(* CODESYS project OC_Profinet.library
   DefaultNamespace: OC_Profinet
   DocFormat: reStructuredText
   Description: Open Commissioning Library for Profinet devices
   Author: SpiraTec AG
   Title: OC_Profinet
   Version: 0.0.1
   Company: Open Commissioning
   Placeholder: OC_Profinet

Project tree, tasks and I/O mapping:
  libraries: OC_Core, * (Open Commissioning); Tc2_Math, * (Beckhoff Automation GmbH); Tc2_Standard, * (Beckhoff Automation GmbH); Tc2_System, * (Beckhoff Automation GmbH); Tc2_Utilities, * (Beckhoff Automation GmbH); Tc3_Module, * (Beckhoff Automation GmbH); TcUnit, * (www.tcunit.org)
  Common/
    ProfidriveBaseState/
    ProfidriveParamInterpreter/
      data type E_ProfidriveParamFormat
      function block FB_ProfidriveParamInterpreter [ST]: FormatSize, FormatType, MakeResponse, Reset
      data type ST_ProfidriveParam
      data type ST_ProfidriveParamSet
  Devices/
    Communication/
      RcvDp/
        function block FB_RcvDp [ST]: AssignProcessData, ControlLogic, InitRun, ReadBus, SimLogic, WriteBus
        data type ST_RcvDpConfig
        data type ST_RcvDpCtrl
        data type ST_RcvDpDevData
        data type ST_RcvDpHstData
        data type ST_RcvDpStatus
      SendDp/
        function block FB_SendDp [ST]: AssignProcessData, ControlLogic, InitRun, PlcAddress, ReadBus, SimLogic, WriteBus
        data type ST_SendDpConfig
        data type ST_SendDpCtrl
        data type ST_SendDpDevData
        data type ST_SendDpHstData
        data type ST_SendDpStatus
      function F_CalcCrc16 [ST]
    Drives/
      MoviCPosition/
        data type E_MoviCPositionOperationMode
        function block FB_MoviCPosition [ST]: AssignProcessData, ControlLogic, GetControlData, InitRun, Operation, Safety, SetStatusData
        data type ST_MoviCPosition_Config
        data type ST_MoviCPosition_Control
        data type ST_MoviCPosition_Status
      MoviCVelocity/
        function block FB_MoviCVelocity [ST]: AssignProcessData, ControlLogic, GetControlData, InitRun, Operation, Safety, SetStatusData
        data type ST_MoviCVelocity_Config
        data type ST_MoviCVelocity_Control
        data type ST_MoviCVelocity_Status
      MovisafeCSBx1a/
        function block FB_MovisafeCSBx1a [ST]: AssignProcessData, ControlLogic, GetControlData, InitRun, SetStatusData
        data type ST_MovisafeCSBx1a_Config
        data type ST_MovisafeCSBx1a_Control
        data type ST_MovisafeCSBx1a_Status
      MovisafeCSSx1a/
        function block FB_MovisafeCSSx1a [ST]: AssignProcessData, ControlLogic, GetControlData, InitRun, SetStatusData
        data type ST_MovisafeCSSx1a_Config
        data type ST_MovisafeCSSx1a_Control
        data type ST_MovisafeCSSx1a_Status
      ProfidriveGSM/
        data type E_ProfidriveGSM_State
        function block FB_ProfidriveGSM [ST]: eState, nControl, nStatus, S0_Disabled, S1_SwitchingOnInhibited, S2_ReadyForSwitchingOn, S3_SwitchedOn, S4_Operation, S51_RampStop, S52_QuickStop
        data type ST_ProfiidriveGSM_STW1
        data type ST_ProfiidriveGSM_ZSW1
      ProfidriveTelegram1/
        function block FB_ProfidriveTelegram1 [ST]: AssignProcessData, ControlLogic, GetControlData, InitRun, Operation, SetStatusData
        data type ST_ProfidriveTelegram1_Config
        data type ST_ProfidriveTelegram1_Control
        data type ST_ProfidriveTelegram1_Status
  Tests/
    Drives/
      function block FB_ProfidriveGSM_Test [ST]: TestState_S0, TestState_S1, TestState_S2, TestState_S3, TestState_S4, TestState_S51, TestState_S52, TestTransitions_S0, TestTransitions_S1, TestTransitions_S2, TestTransitions_S3, TestTransitions_S4, TestTransitions_S51, TestTransitions_S52
      function block FB_ProfidriveTelegram1_Test [ST]: Test_ProcessDataControl, Test_ProcessDataStatus
    program PRG_TEST [ST]
*)

// Common/ProfidriveParamInterpreter/E_ProfidriveParamFormat
{attribute 'qualified_only'}
{attribute 'strict'}
{attribute 'conditionalshow'}
TYPE E_ProfidriveParamFormat :
(
	UNKNOWN := 0,
	INT8	:= 2,
	INT16	:= 3,
	INT32	:= 4,
	UINT8	:= 5,
	UINT16	:= 6,
	UINT32	:= 7,
	FLOAT	:= 8,
	ZERO	:= 64,
	BYTE_	:= 65,
	WORD_	:= 66,
	DWORD_	:= 67,
	ERROR	:= 68
) BYTE;
END_TYPE

// Common/ProfidriveParamInterpreter/ST_ProfidriveParam
{attribute 'conditionalshow'}
TYPE ST_ProfidriveParam :
STRUCT
	nAttribute	: BYTE;
	nNumber		: UINT;
	nSubIndex	: UINT;
	nElements	: BYTE;
	nFormat		: E_ProfidriveParamFormat;
	aValue		: ARRAY[0..234] OF BYTE;
END_STRUCT
END_TYPE

// Common/ProfidriveParamInterpreter/ST_ProfidriveParamSet
{attribute 'conditionalshow'}
TYPE ST_ProfidriveParamSet :
	ARRAY[0..22] OF ST_ProfidriveParam; 
END_TYPE

// Devices/Communication/RcvDp/ST_RcvDpConfig
TYPE ST_RcvDpConfig :
STRUCT
	nDpDpId			 			: UINT := 0;
	fTimeout		 			: REAL := 0.5;
	bAutoAckRei					: BOOL := TRUE;
END_STRUCT
END_TYPE

// Devices/Communication/RcvDp/ST_RcvDpCtrl
{attribute 'pack_mode' := '1'}
TYPE ST_RcvDpCtrl :
STRUCT
	nRcvBoolData			: WORD;
	nRcvInt00				: INT;
	nRcvInt01				: INT;
	nRcvData				: WORD;
	nRcvSequenceNumber		: WORD;
	nRcvCrc					: WORD;
END_STRUCT
END_TYPE

// Devices/Communication/RcvDp/ST_RcvDpDevData
TYPE ST_RcvDpDevData :
STRUCT
	bAckRei		: BOOL;
	bSub00		: BOOL;
	bSub01		: BOOL;
	bSub02		: BOOL;
	bSub03		: BOOL;
	bSub04		: BOOL;
	bSub05		: BOOL;
	bSub06		: BOOL;
	bSub07		: BOOL;
	bSub08		: BOOL;
	bSub09		: BOOL;
	bSub10		: BOOL;
	bSub11		: BOOL;
	bSub12		: BOOL;
	bSub13		: BOOL;
	bSub14		: BOOL;
	bSub15		: BOOL;
	nSub00		: INT;
	nSub01		: INT;
END_STRUCT
END_TYPE

// Devices/Communication/RcvDp/ST_RcvDpHstData
TYPE ST_RcvDpHstData :
STRUCT
	bError		: BOOL;
	bSubsOn		: BOOL;
	bRcv00		: BOOL;
	bRcv01		: BOOL;
	bRcv02		: BOOL;
	bRcv03		: BOOL;
	bRcv04		: BOOL;
	bRcv05		: BOOL;
	bRcv06		: BOOL;
	bRcv07		: BOOL;
	bRcv08		: BOOL;
	bRcv09		: BOOL;
	bRcv10		: BOOL;
	bRcv11		: BOOL;
	bRcv12		: BOOL;
	bRcv13		: BOOL;
	bRcv14		: BOOL;
	bRcv15		: BOOL;
	nRcv00		: INT;
	nRcv01		: INT;
END_STRUCT
END_TYPE

// Devices/Communication/RcvDp/ST_RcvDpStatus
{attribute 'pack_mode' := '1'}
TYPE ST_RcvDpStatus :
STRUCT
	nSendData				: WORD;
	nSendSequenceNumber		: WORD;	
	nSendCrc				: WORD;
END_STRUCT
END_TYPE

// Devices/Communication/SendDp/ST_SendDpConfig
TYPE ST_SendDpConfig :
STRUCT
	nDpDpId			 			: UINT := 0;
	fTimeout		 			: REAL := 0.5;
END_STRUCT
END_TYPE

// Devices/Communication/SendDp/ST_SendDpCtrl
TYPE ST_SendDpCtrl :
STRUCT
	nRcvData				: WORD;
	nRcvSequenceNumber		: WORD;	
	nRcvCrc					: WORD;
END_STRUCT
END_TYPE

// Devices/Communication/SendDp/ST_SendDpDevData
TYPE ST_SendDpDevData :
STRUCT
	bSend00		: BOOL;
	bSend01		: BOOL;
	bSend02		: BOOL;
	bSend03		: BOOL;
	bSend04		: BOOL;
	bSend05		: BOOL;
	bSend06		: BOOL;
	bSend07		: BOOL;
	bSend08		: BOOL;
	bSend09		: BOOL;
	bSend10		: BOOL;
	bSend11		: BOOL;
	bSend12		: BOOL;
	bSend13		: BOOL;
	bSend14		: BOOL;
	bSend15		: BOOL;
	nSend00		: INT;
	nSend01		: INT;
END_STRUCT
END_TYPE

// Devices/Communication/SendDp/ST_SendDpHstData
TYPE ST_SendDpHstData :
STRUCT
	bError		: BOOL;
	bSubsOn		: BOOL;
END_STRUCT
END_TYPE

// Devices/Communication/SendDp/ST_SendDpStatus
TYPE ST_SendDpStatus :
STRUCT
	nSendBoolData			: WORD;
	nSendInt00				: INT;
	nSendInt01				: INT;
	nSendData				: WORD;
	nSendSequenceNumber		: WORD;
	nSendCrc				: WORD;
END_STRUCT
END_TYPE

// Devices/Drives/MoviCPosition/E_MoviCPositionOperationMode
{attribute 'qualified_only'}
TYPE E_MoviCPositionOperationMode :
(
	Jog					:= 100, //Position controlled jogging
	JogNoEnc			:= 101, //Speed controlled jogging
	SpeedControl		:= 200, //Speed control
	ReferenceParam		:= 300, //Reference travel, offset via parameter
	ReferenceBus		:= 301, //Reference travel, offset via fieldbus
	PositionAbs			:= 400, //Absolute position control
	PositionRel			:= 401, //Relative position control
	PositionModPos		:= 402, //Modulo position control, positive
	PositionModNeg		:= 403, //Modulo position control, negative
	PositionModShort	:= 404, //Modulo position control, shortest distance
	EnergyOptimized		:= 1200, //Energieoptimiertes Positionieren
	MechanicsOptimized	:= 1210	 //Mechanikoptimiertes Positionieren
)INT;
END_TYPE

// Devices/Drives/MoviCPosition/ST_MoviCPosition_Config
TYPE ST_MoviCPosition_Config :
STRUCT
	pMovisafeCSSx1a			: POINTER TO FB_MovisafeCSSx1a; //[optional] Pointer to a MovisafeCSSx1a instance
	nSoftwareLimitMin		: DINT := -2147483648;	//Position limit minimum in LU
	nSoftwareLimitMax		: DINT := 2147483647;	//Position limit maximum in LU
	nReferencePos			: DINT := 0;			//Reference position in LU when using mode 300
	fDecCoastStop			: REAL := 1000.0;		//Deceleration for coast/brake stop in LU/s^2
	fDecEstop				: REAL := 100.0;		//Deceleration for emergency stop in LU/s^2
	fDecelerationLimit		: REAL := 100.0;		//Decceleration limit (bus stop) in LU/s^2
	fRatioVelocity			: REAL := 1.0;			//Ratio for setpoint velocity
	fRatioAccDec			: REAL := 1.0;			//Ratio for setpoint acceleration/deceleration
	fRatioPosition			: REAL := 1.0;			//Ratio for position output
	nJerk					: INT  := 0;			//Jerk from 0 to 100%
	fPositionOffset			: REAL := 0;
	fInitPosition			: REAL := 0;
	fResolution				: REAL := 0.1;
	bSwapProcessData		: BOOL; //SWAP Process Data from/to FIELDBUS
END_STRUCT
END_TYPE

// Devices/Drives/MoviCPosition/ST_MoviCPosition_Control
{attribute 'pack_mode' := '1'}
TYPE ST_MoviCPosition_Control :
STRUCT
    b0_EnableEStop 					: BIT;	//0  1 = enable, 0 = emergency stop
    b1_EnableBusStop 				: BIT;	//1  1 = enable, 0 = stop at application limits
    b2_Reserved2 					: BIT;	//2
    b3_ReleaseBrake 				: BIT;	//3  only needed if function is activated
    b4_JoggingCW 					: BIT;	//4  jog positive
    b5_JoggingCCW 					: BIT;	//5  jog negative
    b6_AcceptRelativePosition 		: BIT;	//6  apply relative target pos only in relative pos mode
    b7_StartStop 					: BIT;	//7  1 = start movement in all modes except jog, 0 = deceleration to speed 0
    b8_ErrorReset 					: BIT;	//8  reset fault messages
    b9_Reserved9 					: BIT;	//9
    b10_ActivateDriveTrain2 		: BIT;	//10  0 = drive train 1 selected, 1 = drive train 2 selected
    b11_Reserved11 					: BIT;	//11
    b12_DisableSoftwareLimits 		: BIT;	//12  0 = software limit activated, 1 = software limit deactivated
    b13_ActivateInhibit 			: BIT;	//13  1 = output stage inhibit activated -> motor coasts to halt or brake is applied, 0 = output stage can be enabled
    b14_ActivateStandByMode 		: BIT;	//14  1 = activated, can only be activated when output stage is inhibited (bActivateInhibit = 1)
    b15_MovikitHeartbeat 			: BIT;	//15  Heartbeat trigger
	nSetpointSpeed					: INT;	//16..31 
	nSetpointAcceleration			: INT;	//32..47
	nSetpointDeceleration			: INT;	//48..63
	nDigitalOutputs					: WORD;	//64..79
	nTargetApplicationMode			: E_MoviCPositionOperationMode; //80..95
	nTargetPosition					: DINT;	//96..127
END_STRUCT
END_TYPE

// Devices/Drives/MoviCPosition/ST_MoviCPosition_Status
{attribute 'pack_mode' := '1'}
TYPE ST_MoviCPosition_Status :
STRUCT
	b0_InverterReady					: BIT;	//0  1 = Ready
	b1_STOInactive						: BIT;	//1  1 = STO inactive
	b2_PowerStageOn						: BIT;	//2  1 = Output stage enable
	b3_BrakeReleased					: BIT;	//3  1 = Brake released
	b4_MotorTurning						: BIT;	//4  1 = Motor running
	b5_DriveReferenced					: BIT;	//5  1 = Active drive referenced
	b6_SetpointsActive					: BIT;	//6  1 = New relative position applied
	b7_TargetpositionReached			: BIT;	//7  1 = In position
	b8_ErrorActive						: BIT;	//8  1 = Fault
	b9_WarningActive					: BIT;	//9  1 = Warning
	b10_DriveTrain2Active				: BIT;	//10  1 = Drive train 2 active
	b11_SpeedSetpointReached			: BIT;	//11  1 = "Setpoint/actual speed comparison active" signal
	b12_SoftwareLimitsDisabled			: BIT;	//12  1 = Software limit switches inactive
	b13_OutputStageInhibit 				: BIT;	//13  1 = Output stage inhibit 
	b14_StandByModeActive				: BIT;	//14  1 = Standby mode active
	b15_MovikitHeartbeat				: BIT;	//15  Heartbeat trigger mirror
	nActualSpeed						: INT;	//16..31
	nActualStatus						: WORD;	//32..47
	nActualTorque						: INT;	//48..63
	nDigitalInputs						: WORD;	//64..79
	nActualApplicationMode				: E_MoviCPositionOperationMode; //80..95
	nActualPosition						: DINT;	//96..127 
END_STRUCT
END_TYPE

// Devices/Drives/MoviCVelocity/ST_MoviCVelocity_Config
TYPE ST_MoviCVelocity_Config :
STRUCT
	pMovisafeCSSx1a			: POINTER TO FB_MovisafeCSSx1a; //[optional] Pointer to a MovisafeCSSx1a instance
	nSoftwareLimitMin		: DINT := -2147483648;	//Position limit minimum in LU
	nSoftwareLimitMax		: DINT := 2147483647;	//Position limit maximum in LU
	nReferencePos			: DINT := 0;			//Reference position in LU when using mode 300
	fDecCoastStop			: REAL := 1000.0;		//Deceleration for coast/brake stop in LU/s^2
	fDecEstop				: REAL := 100.0;		//Deceleration for emergency stop in LU/s^2
	fDecelerationLimit		: REAL := 100.0;		//Decceleration limit (bus stop) in LU/s^2
	fRatioVelocity			: REAL := 1.0;			//Ratio for setpoint velocity
	fRatioAccDec			: REAL := 1.0;			//Ratio for setpoint acceleration/deceleration
	fRatioPosition			: REAL := 1.0;			//Ratio for position output
	nJerk					: INT  := 0;			//Jerk from 0 to 100%
	fPositionOffset			: REAL := 0;
	fInitPosition			: REAL := 0;
	fResolution				: REAL := 0.1;
	bSwapProcessData		: BOOL; //SWAP Process Data from/to FIELDBUS
	bOutputVelocity			: BOOL := TRUE;		//TRUE: TargetValue = Velocity, FALSE: TargetValue = Position
END_STRUCT
END_TYPE

// Devices/Drives/MoviCVelocity/ST_MoviCVelocity_Control
TYPE ST_MoviCVelocity_Control :
STRUCT
    b0_EnableEStop 					: BIT;	//0  1 = enable, 0 = emergency stop
    b1_EnableBusStop 				: BIT;	//1  1 = enable, 0 = stop at application limits
    b2_Reserved2 					: BIT;	//2
    b3_ReleaseBrake 				: BIT;	//3  only needed if function is activated
    b4_JoggingCW 					: BIT;	//4  jog positive
    b5_JoggingCCW 					: BIT;	//5  jog negative
    b6_AcceptRelativePosition 		: BIT;	//6  apply relative target pos only in relative pos mode
    b7_StartStop 					: BIT;	//7  1 = start movement in all modes except jog, 0 = deceleration to speed 0
    b8_ErrorReset 					: BIT;	//8  reset fault messages
    b9_Reserved9 					: BIT;	//9
    b10_ActivateDriveTrain2 		: BIT;	//10  0 = drive train 1 selected, 1 = drive train 2 selected
    b11_Reserved11 					: BIT;	//11
    b12_DisableSoftwareLimits 		: BIT;	//12  0 = software limit activated, 1 = software limit deactivated
    b13_ActivateInhibit 			: BIT;	//13  1 = output stage inhibit activated -> motor coasts to halt or brake is applied, 0 = output stage can be enabled
    b14_ActivateStandByMode 		: BIT;	//14  1 = activated, can only be activated when output stage is inhibited (bActivateInhibit = 1)
    b15_MovikitHeartbeat 			: BIT;	//15  Heartbeat trigger
	nSetpointSpeed					: INT;	//16..31 
	nSetpointAcceleration			: INT;	//32..47
	nSetpointDeceleration			: INT;	//48..63
	nDigitalOutputs					: WORD;	//64..79	
END_STRUCT
END_TYPE

// Devices/Drives/MoviCVelocity/ST_MoviCVelocity_Status
{attribute 'pack_mode' := '1'}
TYPE ST_MoviCVelocity_Status :
STRUCT
	b0_InverterReady					: BIT;	//0  1 = Ready
	b1_STOInactive						: BIT;	//1  1 = STO inactive
	b2_PowerStageOn						: BIT;	//2  1 = Output stage enable
	b3_BrakeReleased					: BIT;	//3  1 = Brake released
	b4_MotorTurning						: BIT;	//4  1 = Motor running
	b5_DriveReferenced					: BIT;	//5  1 = Active drive referenced
	b6_SetpointsActive					: BIT;	//6  1 = New relative position applied
	b7_TargetpositionReached			: BIT;	//7  1 = In position
	b8_ErrorActive						: BIT;	//8  1 = Fault
	b9_WarningActive					: BIT;	//9  1 = Warning
	b10_DriveTrain2Active				: BIT;	//10  1 = Drive train 2 active
	b11_SpeedSetpointReached			: BIT;	//11  1 = "Setpoint/actual speed comparison active" signal
	b12_SoftwareLimitsDisabled			: BIT;	//12  1 = Software limit switches inactive
	b13_OutputStageInhibit 				: BIT;	//13  1 = Output stage inhibit 
	b14_StandByModeActive				: BIT;	//14  1 = Standby mode active
	b15_MovikitHeartbeat				: BIT;	//15  Heartbeat trigger mirror
	nActualSpeed						: INT;	//16..31
	nActualStatus						: WORD;	//32..47
	nActualTorque						: INT;	//48..63
	nDigitalInputs						: WORD;	//64..79	
END_STRUCT
END_TYPE

// Devices/Drives/MovisafeCSBx1a/ST_MovisafeCSBx1a_Config
TYPE ST_MovisafeCSBx1a_Config :
STRUCT	
	bSwapProcessData		: BOOL; //SWAP Process Data from/to FIELDBUS
END_STRUCT
END_TYPE

// Devices/Drives/MovisafeCSBx1a/ST_MovisafeCSBx1a_Control
{attribute 'pack_mode' := '1'}
TYPE ST_MovisafeCSBx1a_Control :
STRUCT
	b0_STO1				: BIT; //Sicher abgeschaltetes Drehmoment
	b1_Reserve			: BIT; //Reserve
	b2_Reserve			: BIT; //Reserve
	b3_Reserve			: BIT; //Reserve
	b4_Reserve			: BIT; //Reserve
	b5_Reserve			: BIT; //Reserve
	bQUIT_F_DI			: BIT; //Quittierung der verriegelten Digitaleingänge
	bQUIT_ERROR			: BIT; //Quittierung der Fehler Sicherheitskarte
	b8_Reserve			: BIT; //Reserve
	b9_Reserve			: BIT; //Reserve
	b10_Reserve			: BIT; //Reserve
	b11_Reserve			: BIT; //Reserve
	b12_Reserve			: BIT; //Reserve
	b13_Reserve			: BIT; //Reserve
	b14_Reserve			: BIT; //Reserve
	b15_Reserve			: BIT; //Reserve
	b16_Reserve			: BIT; //Reserve
	b17_Reserve			: BIT; //Reserve
	b18_SSx1			: BIT; //Antriebssicherheitsfunktion SSx1 deaktivieren
	b19_SSx2			: BIT; //Antriebssicherheitsfunktion SSx2 deaktivieren
	b20_Reserve			: BIT; //Reserve
	b21_Reserve			: BIT; //Reserve
	b22_Reserve			: BIT; //Reserve
	b23_Reserve			: BIT; //Reserve
END_STRUCT
END_TYPE

// Devices/Drives/MovisafeCSBx1a/ST_MovisafeCSBx1a_Status
{attribute 'pack_mode' := '1'}
TYPE ST_MovisafeCSBx1a_Status :
STRUCT
	b0_STO_ACTIVE		: BIT; //Sicher abgeschaltetes Drehmoment
	b1_Reserve			: BIT; //Reserve
	b2_Reserve			: BIT; //Reserve
	b3_INPUT_DATA_VALID	: BIT; //Alle Prozesswerte der F-DI enthalten aktuelle Werte
	b4_Reserve			: BIT; //Reserve
	b5_Reserve			: BIT; //Reserve
	b6_WARNING			: BIT; //Warnung in der Safety-option
	b7_ERROR_STATE		: BIT; //Fehler in der Safety-option
	b8_F_DI0			: BIT; //Zustand digitaler Eingang 1
	b9_F_DI1			: BIT; //Zustand digitaler Eingang 2
	b10_F_DI2			: BIT; //Zustand digitaler Eingang 3
	b11_F_DI3			: BIT; //Zustand digitaler Eingang 4
	b12_Reserve			: BIT; //Reserve
	b13_Reserve			: BIT; //Reserve
	b14_Reserve			: BIT; //Reserve
	b15_Reserve			: BIT; //Reserve
	b16_Reserve			: BIT; //Reserve
	b17_Reserve			: BIT; //Reserve
	b18_SSx1			: BIT; //SSx1  ist aktiviert
	b19_SSx2			: BIT; //SSx2 ist aktiviert
	b20_Reserve			: BIT; //Reserve
	b21_Reserve			: BIT; //Reserve
	b22_Reserve			: BIT; //Reserve
	b23_Reserve			: BIT; //Reserve
	b24_Reserve			: BIT; //Reserve
	b25_Reserve			: BIT; //Reserve
	b26_Reserve			: BIT; //Reserve
	b27_Reserve			: BIT; //Reserve
	b28_Reserve			: BIT; //Reserve
	b29_Reserve			: BIT; //Reserve
	b30_Reserve			: BIT; //Reserve
	b31_Reserve			: BIT; //Reserve
END_STRUCT
END_TYPE

// Devices/Drives/MovisafeCSSx1a/ST_MovisafeCSSx1a_Config
TYPE ST_MovisafeCSSx1a_Config :
STRUCT	
	bSwapProcessData		: BOOL; //SWAP Process Data from/to FIELDBUS
END_STRUCT
END_TYPE

// Devices/Drives/MovisafeCSSx1a/ST_MovisafeCSSx1a_Control
{attribute 'pack_mode' := '1'}
TYPE ST_MovisafeCSSx1a_Control :
STRUCT
	bSTO				: BIT; //0.0  Sicher abgeschaltetes Drehmoment
	bSLI				: BIT; //0.1  Freigabe SLI (Sicher begrenztes Schrittmaß)
	bSBT				: BIT; //0.2  Freigabe SBT (Sicherer Bremsentest)
	bRES_3				: BIT; //0.3  Reserve
	bMUTING_ENC_ERR		: BIT; //0.4  Muting Geber anwählen
	bTEST_MODE_ACTIVE	: BIT; //0.5  Test Modus der Antriebssicherheitsfunktion anwählen
	bQUIT_F_DI			: BIT; //0.6  Quittierung der verriegelten Digitaleingänge
	bQUIT_ERROR			: BIT; //0.7  Quittierung der Fehler Sicherheitskarte
	bF_DO_0				: BIT; //1.0  F-DO 00 Digitaler Ausgang 0
	bF_DO_1				: BIT; //1.1  F-DO 01 Digitaler Ausgang 1
	bRES_12				: BIT; //1.2  Reserve
	bRES_13				: BIT; //1.3  Reserve
	bRES_14				: BIT; //1.4  Reserve
	bRES_15				: BIT; //1.5  Reserve
	bRES_16				: BIT; //1.6  Reserve
	bRES_17				: BIT; //1.7  Reserve
	bSOS_1				: BIT; //2.0  SOS1 deaktivieren (Sicherer Betriebshalt)
	bRES_21				: BIT; //2.1  Reserve
	bSSx1				: BIT; //2.2  Antriebssicherheitsfunktion SSx1 deaktivieren
	bSSx2				: BIT; //2.3  Antriebssicherheitsfunktion SSx2 deaktivieren
	bSDI_1				: BIT; //2.4  SDI 1 deaktivieren (Sichere Bewegungsrichtung)
	bSDI_2				: BIT; //2.5  SDI 2 deaktivieren (Sichere Bewegungsrichtung)
	bSLI_1				: BIT; //2.6  SLI 1 deaktivieren (Sicher begrenztes Schrittmaß)
	bSLI_2				: BIT; //2.7  SLI 2 deaktivieren (Sicher begrenztes Schrittmaß)
	bSLS_1				: BIT; //3.0  SLS 1 deaktivieren (Sicher begrenzte Geschwindigkeit)
	bSLS_2				: BIT; //3.1  SLS 2 deaktivieren (Sicher begrenzte Geschwindigkeit)
	bSLS_3				: BIT; //3.2  SLS 3 deaktivieren (Sicher begrenzte Geschwindigkeit)
	bSLS_4				: BIT; //3.3  SLS 4 deaktivieren (Sicher begrenzte Geschwindigkeit)
	bSSR_1				: BIT; //3.4  SSR 1 deaktivieren (Sicherer Geschwindigkeitsbereich)
	bSSR_2				: BIT; //3.5  SSR 2 deaktivieren (Sicherer Geschwindigkeitsbereich)
	bRES_36				: BIT; //3.6  Reserve
	bRES_37				: BIT; //3.7  Reserve
	bSLA_1				: BIT; //4.0  SLA 1 deaktivieren (Sicher begrenzte Beschleunigung)
	bSLA_2				: BIT; //4.1  SLA 2 deaktivieren (Sicher begrenzte Beschleunigung)
	bRES_42				: BIT; //4.2  Reserve
	bRES_43				: BIT; //4.3  Reserve
	bRES_44				: BIT; //4.4  Reserve
	bRES_45				: BIT; //4.5  Reserve
	bRES_46				: BIT; //4.6  Reserve
	bRES_47				: BIT; //4.7  Reserve
END_STRUCT
END_TYPE

// Devices/Drives/MovisafeCSSx1a/ST_MovisafeCSSx1a_Status
{attribute 'pack_mode' := '1'}
TYPE ST_MovisafeCSSx1a_Status :
STRUCT
	bSTO_ACTIVE			: BIT; //0.0  Sicher abgeschaltetes Drehmoment
	bASF_DIAG			: BIT; //0.1  Mindestens eine Antriebssicherheitsfunktion hat eine Grenze überschritten
	bSBT_ACTIVE			: BIT; //0.2  Bremsentest ist aktiv
	bINPUT_DATA_VALID	: BIT; //0.3  Alle Prozesswerte der F-DI enthalten aktuelle Werte
	bMUTING_ENC_ERR		: BIT; //0.4  Geber Muting Funktion ist aktive
	bTEST_MODE_ACTIVE	: BIT; //0.5  Test Modus der Antriebssicherheitsfunktion ist aktive
	bWARNING			: BIT; //0.6  Warnung in der Safety-option
	bERROR_STATE		: BIT; //0.7  Fehler in der Safety-option
	bF_DI0				: BIT; //1.0  Zustand digitaler Eingang 1
	bF_DI1				: BIT; //1.1  Zustand digitaler Eingang 2
	bF_DI2				: BIT; //1.2  Zustand digitaler Eingang 3
	bF_DI3				: BIT; //1.3  Zustand digitaler Eingang 4
	bRES_14				: BIT; //1.4  Reserve
	bRES_15				: BIT; //1.5  Reserve
	bRES_16				: BIT; //1.6  Reserve
	bRES_17				: BIT; //1.7  Reserve
	bSOS_1				: BIT; //2.0  SOS1 ist aktiviert (Sicherer Betriebshalt)
	bRES_21				: BIT; //2.1  Reserve
	bSSx1				: BIT; //2.2  SSx1  ist aktiviert
	bSSx2				: BIT; //2.3  SSx2 ist aktiviert
	bSDI_1				: BIT; //2.4  SDI 1  ist aktiviert (Sichere Bewegungsrichtung)
	bSDI_2				: BIT; //2.5  SDI 2  ist aktiviert (Sichere Bewegungsrichtung)
	bSLI_1				: BIT; //2.6  SLI 1  ist aktiviert (Sicher begrenztes Schrittmaß)
	bSLI_2				: BIT; //2.7  SLI 2  ist aktiviert (Sicher begrenztes Schrittmaß)
	bSLS_1				: BIT; //3.0  SLS 1  ist aktiviert (Sicher begrenzte Geschwindigkeit)
	bSLS_2				: BIT; //3.1  SLS 2  ist aktiviert (Sicher begrenzte Geschwindigkeit)
	bSLS_3				: BIT; //3.2  SLS 3  ist aktiviert (Sicher begrenzte Geschwindigkeit)
	bSLS_4				: BIT; //3.3  SLS 4  ist aktiviert (Sicher begrenzte Geschwindigkeit)
	bSSR_1				: BIT; //3.4  SSR 1  ist aktiviert (Sicherer Geschwindigkeitsbereich)
	bSSR_2				: BIT; //3.5  SSR 2  ist aktiviert (Sicherer Geschwindigkeitsbereich)
	bRES_36				: BIT; //3.6  Reserve
	bRES_37				: BIT; //3.7  Reserve
	bSLA_1				: BIT; //4.0  SLA 1  ist aktiviert (Sicher begrenzte Beschleunigung)
	bSLA_2				: BIT; //4.1  SLA 2  ist aktiviert (Sicher begrenzte Beschleunigung)
	bSSM_1				: BIT; //4.2  SSM 1  ist aktiviert (Sichere Geschwindigkeitsüberwachung)
	bSSM_2				: BIT; //4.3  SSM 2  ist aktiviert (Sichere Geschwindigkeitsüberwachung)
	bSSM_3				: BIT; //4.4  SSM 3  ist aktiviert (Sichere Geschwindigkeitsüberwachung)
	bSSM_4				: BIT; //4.5  SSM 4  ist aktiviert (Sichere Geschwindigkeitsüberwachung)
	bRES_46				: BIT; //4.6  Reserve
	bRES_47				: BIT; //4.7  Reserve
	bRES_50				: BIT; //5.0  Reserve
	bRES_51				: BIT; //5.1  Reserve
	bRES_52				: BIT; //5.2  Reserve
	bRES_53				: BIT; //5.3  Reserve
	bRES_54				: BIT; //5.4  Reserve
	bRES_55				: BIT; //5.5  Reserve
	bRES_56				: BIT; //5.6  Reserve
	bRES_57				: BIT; //5.7  Reserve
END_STRUCT
END_TYPE

// Devices/Drives/ProfidriveGSM/E_ProfidriveGSM_State
{attribute 'qualified_only'}
{attribute 'strict'}
{attribute 'conditionalshow'}
TYPE E_ProfidriveGSM_State :
(
	S0_Disabled := 0,
	S1_SwitchingOnInhibited := 1,
	S2_ReadyForSwitchingOn := 2,
	S3_SwitchedOn := 3,
	S4_Operation := 4,
	S51_RampStop := 51,
	S52_QuickStop := 52
);
END_TYPE

// Devices/Drives/ProfidriveGSM/ST_ProfiidriveGSM_STW1
{attribute 'pack_mode' := '1'}
TYPE ST_ProfiidriveGSM_STW1 :
STRUCT
	b0_On 							: BIT; 	//ON/OFF (OFF1)
	b1_CoastStop					: BIT; 	//The axis will not coast stop if this bit is set (OFF2)
	b2_QuickStop					: BIT; 	//The axis will not execute quick stop if this bit is set. Quick stop executes a controlled stop on the axis. (OFF3)
	b3_EnableOperation				: BIT; 	//The axis will enable and execute command if all preconditions are set. If a Wake and Shake procedure has to be executed as part of enabling, the transition to state "S4: Operation Enabled" is delayed until the procedure is finished.
	b4_Reserve						: BIT;	//Reserve
	b5_Reserve						: BIT;	//Reserve
	b6_Reserve						: BIT;	//Reserve
	b7_FaultAcknowledge				: BIT;	//Set this bit to reset faults on the drive.
	b8_Reserve						: BIT;	//Reserve
	b9_Reserve						: BIT;	//Reserve	
	b10_ControlPlc					: BIT;	//When not set, no command is accepted from the PLC.	
	b11_Reserved					: BIT;	//Reserve
	b12_Reserved					: BIT;	//Reserve
	b13_Reserved					: BIT;	//Reserve
	b14_Reserved					: BIT;	//Reserve
	b15_Reserved					: BIT;	//Reserve
END_STRUCT
END_TYPE

// Devices/Drives/ProfidriveGSM/ST_ProfiidriveGSM_ZSW1
{attribute 'pack_mode' := '1'}
TYPE ST_ProfiidriveGSM_ZSW1 :
STRUCT
	b0_ReadyToSwitchOn 				: BIT; 	//Ready to switch on
	b1_ReadyForOperation			: BIT; 	//Ready for operation
	b2_OperationEnabled				: BIT; 	//Operation enabled
	b3_FaultPresent					: BIT; 	//A fault is present on the axis
	b4_CoastStop 					: BIT;	//No coast stop is executed (No OFF2 is active)
	b5_QuickStop					: BIT;	//No quick stop is executed (No OFF3 is active)
	b6_SwitchingOnInhibited			: BIT;	//Switch-on inhibit Switching on again is only possible through OFF1 and subsequent ON.
	b7_WarningPresent				: BIT;	//Warning present. The drive is operating. No acknowledgment required
	b8_Reserve						: BIT;	//Reserve
	b9_ControlRequested				: BIT;	//Control requested by the master
	b10_Reserved					: BIT;	//Reserve
	b11_Reserved					: BIT;	//Reserve
	b12_Reserved					: BIT;	//Reserve
	b13_Reserved					: BIT;	//Reserve
	b14_Reserved					: BIT;	//Reserve
	b15_Reserved					: BIT;	//Reserve
END_STRUCT
END_TYPE

// Devices/Drives/ProfidriveTelegram1/ST_ProfidriveTelegram1_Config
TYPE ST_ProfidriveTelegram1_Config :
STRUCT
	fRampDownTimeCoastStop 		: REAL := 1.0;		//Coast stop deceleration time in s
	bControlRequested			: BOOL := TRUE;
	bOutputVelocity				: BOOL := TRUE;		//TRUE: TargetValue = Velocity, FALSE: TargetValue = Position
	fP1058						: REAL := 150.0;	//JOG 1 velocity in rotation/s
	fP1059						: REAL := -150.0;	//JOG 1 velocity in rotation/s
	fP1120						: REAL := 2.0;		//Default acceleration time in s
	fP1121						: REAL := 2.0;		//Default deceleration time in s
	fP1135						: REAL := 1.0;		//Ramp down time quick stop in s
	fP2000						: REAL := 3000;		//Velocity in rotation/s when targeting 16#4000
	nR0035						: REAL := 60.0; 	//Temperature in degree celcius	
	bSwapProcessData			: BOOL; //SWAP Process Data from/to FIELDBUS
END_STRUCT
END_TYPE

// Devices/Drives/ProfidriveTelegram1/ST_ProfidriveTelegram1_Control
TYPE ST_ProfidriveTelegram1_Control :
STRUCT
	b0_OFF1								: BOOL;	//STW1_0	0 = OFF1 (braking with ramp-function generator, then pulse suppression & ready for switching on) | 0 → 1 = ON (pulses can be enabled)
	b1_OFF2								: BOOL;	//STW1_1	0 = OFF2 (immediate pulse suppression and switching on inhibited) | 1 = No OFF2 (enable is possible)
	b2_OFF3								: BOOL;	//STW1_2	0 = OFF3 (braking with the OFF3 ramp p1135, then pulse suppression and switching on inhibited) | 1 = No OFF3 (enable possible) 
	b3_EnableOperation					: BOOL;	//STW1_3	0 = Inhibit operation (suppress pulses) | 1 = Enable operation (pulses can be enabled) 
	b4_OperatingCondition				: BOOL;	//STW1_4	0 = Inhibit ramp-function generator (set the ramp-function generator output to zero) | 1 = Operating condition (the ramp-function generator can be enabled)
	b5_ContinueRampFunctionGenerator	: BOOL;	//STW1_5	0 = Freeze ramp-function generator (freeze the ramp-function generator output) | 1 = Continue ramp-function generator 
	b6_EnableSetpoint  					: BOOL;	//STW1_6	0 = Inhibit setpoint (set the ramp-function generator input to zero) | 1 = Enable setpoint 
	b7_AcknowledgeFaults				: BOOL;	//STW1_7	0 → 1: = Acknowledge faults	                            
	b8_Jog1								: BOOL;	//STW1_8	1 = Jog 1 signal source
	b9_Jog2								: BOOL;	//STW1_9	1 = Jog 2 signal source
	b10_ControlByPLC					: BOOL;	//STW1_10	1 = Control by PLC
	b11_SetpointInversion				: BOOL;	//STW1_11	1 = Setpoint inversion
	b12_Reserved						: BOOL;	//STW1_12	Reserved
	b13_PotentiometerSetpointRaise		: BOOL;	//STW1_13	1 = Motorized potentiometer setpoint raise
	b14_PotentiometerSetpointLower		: BOOL;	//STW1_14	1 = Motorized potentiometer setpoint lower
	b15_Reserved						: BOOL;	//STW1_15	Reserved	
	nNSoll 								: INT;
END_STRUCT
END_TYPE

// Devices/Drives/ProfidriveTelegram1/ST_ProfidriveTelegram1_Status
TYPE ST_ProfidriveTelegram1_Status :
STRUCT
	b0_ReadyForSwitchingOn				: BOOL; // ZSW1_0	1 = Ready for switching on
	b1_ReadyForOperation				: BOOL; // ZSW1_1	1 = Ready for operation
	b2_OperationEnabled					: BOOL; // ZSW1_2	1 = Operation enabled
	b3_FaultPresent						: BOOL; // ZSW1_3	1 = Fault present
	b4_NoCoastDownActive				: BOOL; // ZSW1_4	1 = No coast down active (OFF2 inactive)
	b5_NoQuickStopActive				: BOOL; // ZSW1_5	1 = No quick stop active (OFF3 inactive)
	b6_SwitchingOnInhibited				: BOOL; // ZSW1_6	1 = Switching on inhibited active
	b7_AlarmPresent						: BOOL; // ZSW1_7	1 = Alarm present                        	
	b8_DeviationWithinTolerance			: BOOL; // ZSW1_8	1 = Speed setpoint - actual value deviation within tolerance t_off
	b9_ControlRequested					: BOOL; // ZSW1_9	1 = Control requested        
	b10_RpmCompValueReachedOrExceeded	: BOOL; // ZSW1_10	1 = f or n comparison value reached/exceeded  
	b11_TorqueOrPowerLimitNotReached	: BOOL; // ZSW1_11	1 = I, M, or P limit not reached     
	b12_OpenHoldingBrake 				: BOOL; // ZSW1_12	1 = Open the holding brake      
	b13_NoOvertempAlarm					: BOOL; // ZSW1_13	1 = No motor overtemperature alarm      
	b14_MotorRotatesForwards			: BOOL; // ZSW1_14	1 = Motor rotates forwards (n_act >= 0) | 0 = Motor rotates backwards (n_act < 0)   
	b15_NoAlarmNoOvertempPowerUnit		: BOOL; // ZSW1_15	1 = No alarm, thermal overload, power unit  
	nNIst								: INT;
END_STRUCT
END_TYPE

// Common/ProfidriveParamInterpreter/FB_ProfidriveParamInterpreter
FUNCTION_BLOCK INTERNAL FB_ProfidriveParamInterpreter
VAR_INPUT
	(* Pointer to raw user data *)
	pRawData		: POINTER TO BYTE;
	(* Pointer to array of parameters *)
	pParamSet		: POINTER TO ST_ProfidriveParamSet;
END_VAR
VAR_OUTPUT
	(* Reference number for response *)
	nReference		: BYTE;
	(* 1 = read, 2 = write *)
	nCommand		: BYTE;
	(* Addressed axis number *)
	nAxis			: BYTE;
	(* Number of parameters to read/write *)
	nParameters		: BYTE;
END_VAR
VAR
	nOffsReq		: BYTE;
	nOffsValue		: BYTE;
	nFormatSize		: BYTE;
	nValues			: BYTE;
	i, j, k			: UINT;
END_VAR

(* Copy header (first 4 bytes) *)
	nReference := pRawData[0];
	nCommand := pRawData[1];
	nAxis := pRawData[2];
	nParameters := pRawData[3];

(* Set request offset behind header *)
	nOffsReq := 4;

(* Set value offset behind last request *)
	nOffsValue := 4 + nParameters * 6;

(* Reset all parameters *)
	memset(pParamSet, 0, SIZEOF(ST_PROFIdriveParamSet));

(* Check parameter number *)	
	IF nParameters = 0 THEN
		RETURN;
	END_IF

(* Loop through number of parameter requests *)
	FOR i := 0 TO nParameters - 1 BY 1 DO
		
		(* Get parameter request information (6 bytes)... *)
		pParamSet^[i].nAttribute := pRawData[nOffsReq];
		pParamSet^[i].nElements := pRawData[nOffsReq + 1];
		pParamSet^[i].nNumber := pRawData[nOffsReq + 2] * 16#100 + pRawData[nOffsReq + 3];
		pParamSet^[i].nSubIndex := pRawData[nOffsReq + 4] * 16#100 + pRawData[nOffsReq + 5];
		
		(* ... and set offset to next request *)
		nOffsReq := nOffsReq + 6;
				
		(* Write command -> get values *)
		IF nCommand = 2 THEN		
			(* Get format *)
			nFormatSize := FormatSize(pRawData[nOffsValue]);
			pParamSet^[i].nFormat := FormatType(pRawData[nOffsValue]);
			nOffsValue := nOffsValue + 1;
			
			(* Get number of values *)
			nValues := pRawData[nOffsValue];
			nOffsValue := nOffsValue + 1;
			
			(* Loop through number of values *)
			FOR j := 0 TO nValues - 1 BY 1 DO
				
				(* Set value offset behind current values *)
				nOffsValue := nOffsValue + nFormatSize;
				
				(* Loop through format size and get values in reverse order *)
				FOR k := 0 TO nFormatSize - 1 BY 1 DO
					pParamSet^[i].aValue[j + k] := pRawData[nOffsValue - k - 1];
				END_FOR
			END_FOR
			
			(* Check if odd and set to even number *)
			IF nOffsValue.0 THEN
				nOffsValue := nOffsValue + 1;
			END_IF
		END_IF
	END_FOR

METHOD INTERNAL FormatSize : BYTE
VAR_INPUT
	nFormat	: BYTE;
END_VAR
CASE nFormat OF
	 16#02 : FormatSize := 2;
	 16#03 : FormatSize := 2;
	 16#04 : FormatSize := 4;
	 16#05 : FormatSize := 2;
	 16#06 : FormatSize := 2;
	 16#07 : FormatSize := 4;
	 16#08 : FormatSize := 4;
	 16#40 : FormatSize := 0;
	 16#41 : FormatSize := 2;
	 16#42 : FormatSize := 2;
	 16#43 : FormatSize := 4;
	 16#44 : FormatSize := 0;
ELSE
	FormatSize := 0;
END_CASE
END_METHOD

METHOD INTERNAL FormatType : E_ProfidriveParamFormat
VAR_INPUT
	nFormat	: BYTE;
END_VAR
CASE nFormat OF
	 16#02 : FormatType := E_ProfidriveParamFormat.INT8;
	 16#03 : FormatType := E_ProfidriveParamFormat.INT16;
	 16#04 : FormatType := E_ProfidriveParamFormat.INT32;
	 16#05 : FormatType := E_ProfidriveParamFormat.UINT8;
	 16#06 : FormatType := E_ProfidriveParamFormat.UINT16;
	 16#07 : FormatType := E_ProfidriveParamFormat.UINT32;
	 16#08 : FormatType := E_ProfidriveParamFormat.FLOAT;
	 16#40 : FormatType := E_ProfidriveParamFormat.ZERO;
	 16#41 : FormatType := E_ProfidriveParamFormat.BYTE_;
	 16#42 : FormatType := E_ProfidriveParamFormat.WORD_;
	 16#43 : FormatType := E_ProfidriveParamFormat.DWORD_;
	 16#44 : FormatType := E_ProfidriveParamFormat.ERROR;
ELSE
	FormatType := E_PROFIdriveParamFormat.UNKNOWN;
END_CASE
END_METHOD

METHOD INTERNAL MakeResponse : BOOL
VAR_INPUT
	(* Pointer to acyclic user data *)
	pResData		: POINTER TO BYTE;
END_VAR
VAR
	nOffset			: BYTE;
	nFormatSize		: BYTE;
	i, j, k			: UINT;
END_VAR
(* Copy header (first 4 bytes) *)
	pResData[0] := nReference;
	pResData[1] := nCommand;
	pResData[2] := nAxis;
	pResData[3] := nParameters;

(* Set offset behind header *)
	nOffset := 4;
	
(* Check parameter number *)	
	IF nParameters = 0 THEN
		RETURN;
	END_IF

(* Loop through number of parameter requests *)
	FOR i := 0 TO nParameters - 1 BY 1 DO
		
		(* Set format *)
		pResData[nOffset] := pParamSet^[i].nFormat;
		nFormatSize := FormatSize(pParamSet^[i].nFormat);
		nOffset := nOffset + 1;
		
		(* Set number of values *)
		pResData[nOffset] := pParamSet^[i].nElements;
		nOffset := nOffset + 1;
		
		(* Loop through number of elements *)
		FOR j := 0 TO pParamSet^[i].nElements - 1 BY 1 DO
			
			(* Set value offset behind current values *)
			nOffset := nOffset + nFormatSize;
			
			(* Loop through format size and get values in reverse order *)
			
			IF nFormatSize > 0 THEN
				FOR k := 0 TO nFormatSize - 1 BY 1 DO
					pResData[nOffset - k - 1] := pParamSet^[i].aValue[j + k] ;
				END_FOR
			END_IF
			
		END_FOR
		
		(* Check if odd and set to even number *)
		IF nOffset.0 THEN
			nOffset := nOffset + 1;
		END_IF	
	END_FOR

(* Return true when finished *)
	MakeResponse := TRUE;
END_METHOD

METHOD INTERNAL Reset : BOOL
nReference := 0;
nCommand := 0;
nAxis := 0;
nParameters := 0;
memset(pParamSet, 0, SIZEOF(ST_ProfidriveParamSet));
END_METHOD

END_FUNCTION_BLOCK

// Devices/Communication/RcvDp/FB_RcvDp
{attribute 'reflection'} 
FUNCTION_BLOCK FB_RcvDp EXTENDS FB_Base
VAR_INPUT
	stDevData			: ST_RcvDpDevData;
	stConfig 			: ST_RcvDpConfig;
END_VAR

VAR_OUTPUT
	stHstData			: ST_RcvDpHstData;
END_VAR

VAR
    {attribute 'instance-path'} 
    {attribute 'noinit'} 
    sPath 				: STRING; 
	pControlData		: POINTER TO BYTE;
	pStatusData			: POINTER TO BYTE;
	stCtrl				: ST_RcvDpCtrl; 
	stStatus			: ST_RcvDpStatus; 
	nLastSequenceNumber	: WORD;
	nCalculatedCrc		: WORD;	
	TonTimeout			: TON;	
END_VAR

VAR CONSTANT
	nPolynom			: WORD := 16#4EAB;
END_VAR

SUPER^();
InitRun();	
ReadBus();
ControlLogic();
WriteBus();

(*Assign Process Data Objects to device*)
METHOD PUBLIC AssignProcessData : BOOL
VAR_INPUT
	aControlData 		: ANY; //Addr. Process Output 12 bytes
	aStatusData 		: ANY; //Addr. Process Input 6 bytes
END_VAR
THIS^.pControlData := aControlData.pValue;
THIS^.pStatusData := aStatusData.pValue;
END_METHOD

METHOD INTERNAL ControlLogic
VAR_INPUT
END_VAR
(* Simplified communication when using PLCSIM Adv. *)
	IF OC_Core.GVL_Core.fbSystem.eControllerType = E_ControllerType.PlcSimAdvanced THEN
		SimLogic();
		RETURN;
	END_IF

(* Calculate received crc *)
	nCalculatedCrc := F_CalcCrc16(ADR(stCtrl), 8, stConfig.nDpDpId, nPolynom);

(* Restart timer, if sequence number has changed *)
	IF stCtrl.nRcvSequenceNumber <> nLastSequenceNumber AND NOT stHstData.bError THEN
		nLastSequenceNumber := stCtrl.nRcvSequenceNumber;
		stHstData.bSubsOn	:= FALSE;
		TonTimeout.IN		:= FALSE;
	ELSE
		TonTimeout.IN		:= TRUE;
	END_IF

(* Reintegration *)
	IF (stConfig.bAutoAckRei AND stHstData.bError) OR stDevData.bAckRei THEN
		stHstData.bError 	:= FALSE;
		TonTimeout.IN		:= FALSE;
	END_IF

(* Check if timer has expired *)
	TonTimeout();
	
	IF TonTimeout.Q	THEN
		stHstData.bError	:= TRUE;
		stHstData.bSubsOn	:= TRUE;
	END_IF

(* compare received crc value with calculated crc *)
	IF stCtrl.nRcvCrc = nCalculatedCrc AND NOT stHstData.bError THEN
		stHstData.bSubsOn	:= FALSE;
	ELSE
		stHstData.bError	:= TRUE;
		stHstData.bSubsOn	:= TRUE;
	END_IF

(* Get substitude or safety values *)
	IF stHstData.bSubsOn THEN
		stHstData.bRcv00	:= stDevData.bSub00;
		stHstData.bRcv01	:= stDevData.bSub01;
		stHstData.bRcv02	:= stDevData.bSub02;
		stHstData.bRcv03	:= stDevData.bSub03;
		stHstData.bRcv04	:= stDevData.bSub04;
		stHstData.bRcv05	:= stDevData.bSub05;
		stHstData.bRcv06	:= stDevData.bSub06;
		stHstData.bRcv07	:= stDevData.bSub07;
		stHstData.bRcv08	:= stDevData.bSub08;
		stHstData.bRcv09	:= stDevData.bSub09;
		stHstData.bRcv10	:= stDevData.bSub10;
		stHstData.bRcv11	:= stDevData.bSub11;
		stHstData.bRcv12	:= stDevData.bSub12;
		stHstData.bRcv13	:= stDevData.bSub13;
		stHstData.bRcv14	:= stDevData.bSub14;
		stHstData.bRcv15	:= stDevData.bSub15;
		stHstData.nRcv00	:= stDevData.nSub00;
		stHstData.nRcv01	:= stDevData.nSub01;
	ELSE
		stHstData.bRcv00	:= stCtrl.nRcvBoolData.0;
		stHstData.bRcv01	:= stCtrl.nRcvBoolData.1;
		stHstData.bRcv02	:= stCtrl.nRcvBoolData.2;
		stHstData.bRcv03	:= stCtrl.nRcvBoolData.3;
		stHstData.bRcv04	:= stCtrl.nRcvBoolData.4;
		stHstData.bRcv05	:= stCtrl.nRcvBoolData.5;
		stHstData.bRcv06	:= stCtrl.nRcvBoolData.6;
		stHstData.bRcv07	:= stCtrl.nRcvBoolData.7;
		stHstData.bRcv08	:= stCtrl.nRcvBoolData.8;  
		stHstData.bRcv09	:= stCtrl.nRcvBoolData.9;  
		stHstData.bRcv10	:= stCtrl.nRcvBoolData.10;  
		stHstData.bRcv11	:= stCtrl.nRcvBoolData.11;  
		stHstData.bRcv12	:= stCtrl.nRcvBoolData.12; 
		stHstData.bRcv13	:= stCtrl.nRcvBoolData.13; 
		stHstData.bRcv14	:= stCtrl.nRcvBoolData.14; 
		stHstData.bRcv15	:= stCtrl.nRcvBoolData.15;	
		stHstData.nRcv00	:= stCtrl.nRcvInt00;
		stHstData.nRcv01	:= stCtrl.nRcvInt01;
	END_IF

(* Send data *)
	stStatus.nSendData				:= BOOL_TO_WORD(stHstData.bSubsOn);
	stStatus.nSendSequenceNumber	:= stCtrl.nRcvSequenceNumber;
	stStatus.nSendCrc 				:= F_CalcCrc16(ADR(stStatus.nSendData), 2, stConfig.nDpDpId, nPolynom);
END_METHOD

METHOD INTERNAL InitRun : BOOL
VAR_INST
	bInitRun : BOOL := TRUE;
END_VAR
IF NOT bInitRun THEN RETURN; END_IF
bInitRun := FALSE;

IF pControlData = 0 OR pStatusData = 0 THEN
	ADSLOGSTR(ADSLOG_MSGTYPE_WARN, CONCAT(sPath, ': %s'), 'Plc address not set.');
END_IF

TonTimeout.PT := REAL_TO_TIME(stConfig.fTimeout);
END_METHOD

METHOD INTERNAL ReadBus
VAR_INPUT
END_VAR
IF pControlData = 0 THEN
	RETURN;
END_IF

stCtrl.nRcvBoolData 		:= pControlData[0] + pControlData[1] * 16#100;
stCtrl.nRcvInt00 			:= UINT_TO_INT(pControlData[2] * 16#100 + pControlData[3]);
stCtrl.nRcvInt01 			:= UINT_TO_INT(pControlData[4] * 16#100 + pControlData[5]);
stCtrl.nRcvData 			:= pControlData[6] + pControlData[7] * 16#100;
stCtrl.nRcvSequenceNumber 	:= pControlData[8] * 16#100 + pControlData[9];
stCtrl.nRcvCrc 				:= pControlData[10] * 16#100 + pControlData[11];
END_METHOD

METHOD INTERNAL SimLogic
VAR_INPUT
END_VAR
(* No error or substitude values in sim mode *)
	stHstData.bError 	:= FALSE;
	stHstData.bSubsOn	:= FALSE;

(* Get safety values *)
	stHstData.bRcv00	:= stCtrl.nRcvBoolData.0;
	stHstData.bRcv01	:= stCtrl.nRcvBoolData.1;
	stHstData.bRcv02	:= stCtrl.nRcvBoolData.2;
	stHstData.bRcv03	:= stCtrl.nRcvBoolData.3;
	stHstData.bRcv04	:= stCtrl.nRcvBoolData.4;
	stHstData.bRcv05	:= stCtrl.nRcvBoolData.5;
	stHstData.bRcv06	:= stCtrl.nRcvBoolData.6;
	stHstData.bRcv07	:= stCtrl.nRcvBoolData.7;
	stHstData.bRcv08	:= stCtrl.nRcvBoolData.8;  
	stHstData.bRcv09	:= stCtrl.nRcvBoolData.9;  
	stHstData.bRcv10	:= stCtrl.nRcvBoolData.10;  
	stHstData.bRcv11	:= stCtrl.nRcvBoolData.11;  
	stHstData.bRcv12	:= stCtrl.nRcvBoolData.12; 
	stHstData.bRcv13	:= stCtrl.nRcvBoolData.13; 
	stHstData.bRcv14	:= stCtrl.nRcvBoolData.14; 
	stHstData.bRcv15	:= stCtrl.nRcvBoolData.15;	
	stHstData.nRcv00	:= stCtrl.nRcvInt00;
	stHstData.nRcv01	:= stCtrl.nRcvInt01;

(* Send data *)
	stStatus.nSendData				:= 16#80;
	stStatus.nSendSequenceNumber	:= stCtrl.nRcvSequenceNumber;
	stStatus.nSendCrc 				:= F_CalcCrc16(ADR(stStatus.nSendData), 2, stConfig.nDpDpId, nPolynom);
END_METHOD

METHOD INTERNAL WriteBus
VAR_INPUT
END_VAR
IF pStatusData = 0 THEN
	RETURN;
END_IF

memcpy(pStatusData, ADR(stStatus.nSendData), 2);
       
memcpy(pStatusData + 2, ADR(stStatus.nSendSequenceNumber) + 1, 1);
memcpy(pStatusData + 3, ADR(stStatus.nSendSequenceNumber), 1);
       
memcpy(pStatusData + 4, ADR(stStatus.nSendCrc) + 1, 1);
memcpy(pStatusData + 5, ADR(stStatus.nSendCrc), 1);
END_METHOD

END_FUNCTION_BLOCK

// Devices/Communication/F_CalcCrc16
FUNCTION F_CalcCrc16 : WORD
VAR_INPUT
	pData		: POINTER TO BYTE;
	nDataSize	: INT;
	nInitCRC	: WORD;
	nPolynom	: WORD;
END_VAR
VAR
	nCrc		: WORD;
	nDataX		: BYTE;
	nI			: INT;
	nJ			: INT;
END_VAR

nCrc := nInitCRC;

FOR nI := 0 TO nDataSize - 1 BY 1 DO
	nDataX	:= pData[nI];
	FOR nJ := 0 TO 7 BY 1 DO
		IF (SHR(nCrc,15) AND 1) <> (SHR(nDataX,7) AND 1) THEN
			nCrc := SHL(nCrc,1) XOR nPolynom;
		ELSE
			nCrc := SHL(nCrc,1);
		END_IF
		nDataX := SHL(nDataX,1);
	END_FOR	
END_FOR

F_CalcCrc16 := nCrc;

END_FUNCTION

// Devices/Communication/SendDp/FB_SendDp
{attribute 'reflection'} 
FUNCTION_BLOCK FB_SendDp EXTENDS FB_Base
VAR_INPUT
	stDevData			: ST_SendDpDevData;
	stConfig 			: ST_SendDpConfig;
END_VAR

VAR_OUTPUT
	stHstData			: ST_SendDpHstData;
END_VAR

VAR
    {attribute 'instance-path'} 
    {attribute 'noinit'} 
    sPath 				: STRING; 
	pControlData			: POINTER TO BYTE;
	pStatusData				: POINTER TO BYTE;
	stCtrl				: ST_SendDpCtrl; 
	stStatus			: ST_SendDpStatus; 
	nLastSequenceNumber	: WORD;
	nSendSequenceNumber	: WORD;
	nCalculatedCrc		: WORD;	
	TonTimeout			: TON;
END_VAR

VAR CONSTANT
	nPolynom			: WORD := 16#4EAB;
END_VAR

SUPER^();
InitRun();
ReadBus();
ControlLogic();
WriteBus();

(*Assign Process Data Objects to device*)
METHOD PUBLIC AssignProcessData : BOOL
VAR_INPUT
	aControlData 		: ANY; //Addr. Process Output 6 bytes
	aStatusData 		: ANY; //Addr. Process Input 12 bytes
END_VAR
THIS^.pControlData := aControlData.pValue;
THIS^.pStatusData := aStatusData.pValue;
END_METHOD

METHOD INTERNAL ControlLogic
(* Simplified communication when using PLCSIM Adv. *)
	IF OC_Core.GVL_Core.fbSystem.eControllerType = E_ControllerType.PlcSimAdvanced THEN
		SimLogic();
		RETURN;
	END_IF

(* Calculate received crc *)
	nCalculatedCrc := F_CalcCrc16(ADR(stCtrl), 2, stConfig.nDpDpId, nPolynom);

(* Restart timer, if sequence number has changed *)
	IF stCtrl.nRcvSequenceNumber <> nLastSequenceNumber THEN
		TonTimeout.IN		:= FALSE;
		nLastSequenceNumber := stCtrl.nRcvSequenceNumber;
		stHstData.bError	:= FALSE;
		stHstData.bSubsOn	:= FALSE;
	ELSE
		TonTimeout.IN		:= TRUE;
	END_IF

(* Check if timer has expired *)
	TonTimeout();
	
	IF TonTimeout.Q	THEN
		TonTimeout.IN		:= FALSE;
		nSendSequenceNumber := 0;
		stHstData.bError	:= TRUE;
		stHstData.bSubsOn	:= TRUE;
	END_IF

(* compare received crc value with calculated crc *)
	IF stCtrl.nRcvCrc = nCalculatedCrc THEN
		IF nSendSequenceNumber = stCtrl.nRcvSequenceNumber THEN
			IF nSendSequenceNumber = 0 THEN
				nSendSequenceNumber := 1;
			ELSE
				nSendSequenceNumber := nSendSequenceNumber + 1;
			END_IF
		END_IF
	END_IF

(* Limit sequence number to 32767 *)
	IF nSendSequenceNumber > 32767 THEN
		nSendSequenceNumber := 1;
	END_IF

(* Send data *)
	stStatus.nSendBoolData.0 		:= stDevData.bSend00;
	stStatus.nSendBoolData.1 		:= stDevData.bSend01;
	stStatus.nSendBoolData.2 		:= stDevData.bSend02;
	stStatus.nSendBoolData.3 		:= stDevData.bSend03;
	stStatus.nSendBoolData.4 		:= stDevData.bSend04;
	stStatus.nSendBoolData.5 		:= stDevData.bSend05;
	stStatus.nSendBoolData.6 		:= stDevData.bSend06;
	stStatus.nSendBoolData.7 		:= stDevData.bSend07;
	stStatus.nSendBoolData.8 		:= stDevData.bSend08;
	stStatus.nSendBoolData.9 		:= stDevData.bSend09;
	stStatus.nSendBoolData.10 		:= stDevData.bSend10;
	stStatus.nSendBoolData.11 		:= stDevData.bSend11;
	stStatus.nSendBoolData.12 		:= stDevData.bSend12;
	stStatus.nSendBoolData.13 		:= stDevData.bSend13;
	stStatus.nSendBoolData.14 		:= stDevData.bSend14;
	stStatus.nSendBoolData.15 		:= stDevData.bSend15;
	stStatus.nSendInt00				:= stDevData.nSend00;
	stStatus.nSendInt01				:= stDevData.nSend01;
	stStatus.nSendData				:= BOOL_TO_WORD(stHstData.bSubsOn);
	stStatus.nSendSequenceNumber 	:= nSendSequenceNumber;
	stStatus.nSendCrc 				:= F_CalcCrc16(ADR(stStatus), 8, stConfig.nDpDpId, nPolynom);
END_METHOD

METHOD INTERNAL InitRun : BOOL
VAR_INST
	bInitRun : BOOL := TRUE;
END_VAR
IF NOT bInitRun THEN RETURN; END_IF
bInitRun := FALSE;

IF pControlData = 0 OR pStatusData = 0 THEN
	ADSLOGSTR(ADSLOG_MSGTYPE_WARN, CONCAT(sPath, ': %s'), 'Plc address not set.');
END_IF

TonTimeout.PT := REAL_TO_TIME(stConfig.fTimeout);
END_METHOD

METHOD PUBLIC PlcAddress
VAR_INPUT
	I :	ANY; // Must be 6 bytes 
	Q :	ANY; // Must be 12 bytes
END_VAR
pControlData := Q.pValue;
pStatusData := I.pValue;
END_METHOD

METHOD INTERNAL ReadBus
VAR_INPUT
END_VAR
IF pControlData = 0 THEN
	RETURN;
END_IF

stCtrl.nRcvData 			:= pControlData[0] + pControlData[1] * 16#100;
stCtrl.nRcvSequenceNumber 	:= pControlData[2] * 16#100 + pControlData[3];
stCtrl.nRcvCrc 				:= pControlData[4] * 16#100 + pControlData[5];
END_METHOD

METHOD INTERNAL SimLogic
VAR_INPUT
END_VAR
(* No error or substitude values in sim mode *)
	stHstData.bError 	:= FALSE;
	stHstData.bSubsOn	:= FALSE;

(* Send data *)
	stStatus.nSendBoolData.0 		:= stDevData.bSend00;
	stStatus.nSendBoolData.1 		:= stDevData.bSend01;
	stStatus.nSendBoolData.2 		:= stDevData.bSend02;
	stStatus.nSendBoolData.3 		:= stDevData.bSend03;
	stStatus.nSendBoolData.4 		:= stDevData.bSend04;
	stStatus.nSendBoolData.5 		:= stDevData.bSend05;
	stStatus.nSendBoolData.6 		:= stDevData.bSend06;
	stStatus.nSendBoolData.7 		:= stDevData.bSend07;
	stStatus.nSendBoolData.8 		:= stDevData.bSend08;
	stStatus.nSendBoolData.9 		:= stDevData.bSend09;
	stStatus.nSendBoolData.10 		:= stDevData.bSend10;
	stStatus.nSendBoolData.11 		:= stDevData.bSend11;
	stStatus.nSendBoolData.12 		:= stDevData.bSend12;
	stStatus.nSendBoolData.13 		:= stDevData.bSend13;
	stStatus.nSendBoolData.14 		:= stDevData.bSend14;
	stStatus.nSendBoolData.15 		:= stDevData.bSend15;
	stStatus.nSendInt00				:= stDevData.nSend00;
	stStatus.nSendInt01				:= stDevData.nSend01;
	stStatus.nSendData				:= 16#80;
	stStatus.nSendSequenceNumber 	:= 16#FFFF;
	stStatus.nSendCrc 				:= F_CalcCrc16(ADR(stStatus), 8, stConfig.nDpDpId, nPolynom);
END_METHOD

METHOD INTERNAL WriteBus
VAR_INPUT
END_VAR
IF pStatusData = 0 THEN
	RETURN;
END_IF

memcpy(pStatusData, ADR(stStatus.nSendBoolData), 2);
       
memcpy(pStatusData + 2, ADR(stStatus.nSendInt00) + 1, 1);
memcpy(pStatusData + 3, ADR(stStatus.nSendInt00), 1);
       
memcpy(pStatusData + 4, ADR(stStatus.nSendInt01) + 1, 1);
memcpy(pStatusData + 5, ADR(stStatus.nSendInt01), 1);
              
memcpy(pStatusData + 6, ADR(stStatus.nSendData), 2);
              
memcpy(pStatusData + 8, ADR(stStatus.nSendSequenceNumber) + 1, 1);
memcpy(pStatusData + 9, ADR(stStatus.nSendSequenceNumber), 1);
               
memcpy(pStatusData + 10, ADR(stStatus.nSendCrc) + 1, 1);
memcpy(pStatusData + 11, ADR(stStatus.nSendCrc), 1);
END_METHOD

END_FUNCTION_BLOCK

// Devices/Drives/MoviCPosition/FB_MoviCPosition
{attribute 'reflection'}
FUNCTION_BLOCK FB_MoviCPosition EXTENDS FB_LinkDataReal
VAR_INPUT
	bSTO						: BOOL := TRUE;
	stControl 					: ST_MoviCPosition_Control;
	stConfig					: ST_MoviCPosition_Config;
	nDigitalInputs				: WORD;
END_VAR

VAR_OUTPUT
	stStatus					: ST_MoviCPosition_Status;
	fValue						: REAL;
END_VAR

VAR
    {attribute 'instance-path'} 
    {attribute 'noinit'} 
    sPath 						: STRING;	                			
	                			
	fbBaseState					: FB_ProfidriveGSM;
	fbBasicDrive				: FB_DriveControl;
	                				
	bOpModeValid				: BOOL;
	pMovisafe					: POINTER TO FB_MovisafeCSSx1a;	
	
	pControlData				: POINTER TO BYTE; //Addr. Process Output
	pStatusData					: POINTER TO BYTE; //Addr. Process Input
END_VAR

SUPER^();
InitRun();

GetControlData();
Safety();
ControlLogic();
SetStatusData();

(*Assign Process Data Objects to device*)
METHOD PUBLIC AssignProcessData : BOOL
VAR_INPUT
	aControlData 		: ANY; //Addr. Process Output
	aStatusData 		: ANY; //Addr. Process Input
END_VAR
THIS^.pControlData := aControlData.pValue;
THIS^.pStatusData := aStatusData.pValue;
END_METHOD

METHOD INTERNAL ControlLogic
//Unity Init - Load persistent data
IF SUPER^.Status.7 THEN
	IF stConfig.fRatioPosition <> 0 THEN	
		fbBasicDrive.fPosition := SUPER^.StatusData/stConfig.fRatioPosition - stConfig.fPositionOffset;
	ELSE
		fbBasicDrive.fPosition := SUPER^.StatusData - stConfig.fPositionOffset;
	END_IF
END_IF

(* Evaluate incoming operation mode *)
bOpModeValid := FALSE;

CASE stControl.nTargetApplicationMode OF
	E_MoviCPositionOperationMode.Jog:
		bOpModeValid := TRUE;
	E_MoviCPositionOperationMode.JogNoEnc:
		bOpModeValid := TRUE;
	E_MoviCPositionOperationMode.SpeedControl:
		bOpModeValid := TRUE;
	E_MoviCPositionOperationMode.ReferenceParam:
		bOpModeValid := TRUE;
	E_MoviCPositionOperationMode.ReferenceBus:
		bOpModeValid := TRUE;
	E_MoviCPositionOperationMode.PositionAbs, E_MoviCPositionOperationMode.EnergyOptimized, E_MoviCPositionOperationMode.MechanicsOptimized:
		bOpModeValid := TRUE;
	E_MoviCPositionOperationMode.PositionRel:
		bOpModeValid := TRUE;
	E_MoviCPositionOperationMode.PositionModPos:
		bOpModeValid := TRUE;
	E_MoviCPositionOperationMode.PositionModNeg:
		bOpModeValid := TRUE;
	E_MoviCPositionOperationMode.PositionModShort:
		bOpModeValid := TRUE;
END_CASE

(* Base state of the controller *)
fbBaseState.bStandstill := OC_Core.F_Compare(fbBasicDrive.fVelocity, 0, 1E-3);
fbBaseState.stSTW1.b0_On := stControl.b1_EnableBusStop AND fbBaseState.eState <> E_ProfidriveGSM_State.S1_SwitchingOnInhibited;
fbBaseState.stSTW1.b1_CoastStop := NOT stControl.b13_ActivateInhibit AND bSTO;
fbBaseState.stSTW1.b2_QuickStop := stControl.b0_EnableEStop;
fbBaseState.stSTW1.b3_EnableOperation := stControl.b7_StartStop AND bOpModeValid;

fbBaseState();
		
(* Set parameter of basic drive *)
IF stControl.b12_DisableSoftwareLimits THEN
	fbBasicDrive.fPositionLimitMin := -2147483648.0;
	fbBasicDrive.fPositionLimitMax := 2147483647.0;
	fbBasicDrive.fTolerance := 0.1;
ELSE
	fbBasicDrive.fPositionLimitMin := DINT_TO_REAL(stConfig.nSoftwareLimitMin);
	fbBasicDrive.fPositionLimitMax := DINT_TO_REAL(stConfig.nSoftwareLimitMax);
	fbBasicDrive.fTolerance := 0.1;
END_IF
					
(* Evaluate base state *)
CASE fbBaseState.eState OF
	
(* S1, S2 or S3 -> Drive coasts to a stop or brake is applied *)
	E_ProfidriveGSM_State.S1_SwitchingOnInhibited,
	E_ProfidriveGSM_State.S2_ReadyForSwitchingOn,
	E_ProfidriveGSM_State.S3_SwitchedOn:
		fbBasicDrive.Stop(stConfig.fDecCoastStop);

(* S4 -> Evaluate operation mode *)
	E_ProfidriveGSM_State.S4_Operation:
		Operation();

(* S5a -> Drive decelerates with application limit *)
	E_ProfidriveGSM_State.S51_RampStop:
		fbBasicDrive.Stop(stConfig.fDecelerationLimit);
		
(* S5b -> Drive decelerates with emergency stop ramp *)
	E_ProfidriveGSM_State.S52_QuickStop:
	    fbBasicDrive.Stop(stConfig.fDecEstop);
END_CASE
	
(* Status Word *)
stStatus.b0_InverterReady				:= TRUE;
stStatus.b1_STOInactive					:= bSTO;
stStatus.b2_PowerStageOn				:= stControl.b13_ActivateInhibit;
stStatus.b3_BrakeReleased				:= stControl.b1_EnableBusStop OR stControl.b3_ReleaseBrake;
stStatus.b4_MotorTurning				:= NOT fbBaseState.bStandstill;
stStatus.b5_DriveReferenced				:= TRUE;
stStatus.b6_SetpointsActive		 		:= FALSE;
stStatus.b7_TargetpositionReached		:= fbBasicDrive.bIsPositionReached;	
stStatus.b8_ErrorActive					:= FALSE;
stStatus.b9_WarningActive				:= FALSE;
stStatus.b10_DriveTrain2Active			:= stControl.b10_ActivateDriveTrain2;
stStatus.b11_SpeedSetpointReached		:= fbBasicDrive.bIsMoving;
stStatus.b12_SoftwareLimitsDisabled		:= stControl.b12_DisableSoftwareLimits;
stStatus.b13_OutputStageInhibit			:= fbBaseState.stZSW1.b6_SwitchingOnInhibited;
stStatus.b14_StandByModeActive			:= stControl.b14_ActivateStandByMode;
stStatus.b15_MovikitHeartbeat			:= stControl.b15_MovikitHeartbeat;

(* Status values *)
stStatus.nActualSpeed := REAL_TO_INT(fbBasicDrive.fVelocity / stConfig.fRatioVelocity);
stStatus.nActualStatus := 0;
stStatus.nActualTorque := 0;
stStatus.nDigitalInputs := nDigitalInputs;
IF bOpModeValid THEN
	stStatus.nActualApplicationMode := stControl.nTargetApplicationMode;
END_IF
stStatus.nActualPosition := REAL_TO_DINT(fbBasicDrive.fPosition);
	
(* Position output *)
THIS^.ControlData := fbBasicDrive.fPosition * stConfig.fRatioPosition + stConfig.fPositionOffset;
fValue := ControlData;
END_METHOD

METHOD INTERNAL GetControlData : BOOL
IF pControlData <= 0 THEN RETURN; END_IF

(* PO1 Control Word *)
F_Memcpy(ADR(stControl), pControlData, 2, stConfig.bSwapProcessData);
(* PO2 Setpoint Speed *)
F_Memcpy(ADR(stControl) + 2, pControlData + 2, 2, stConfig.bSwapProcessData);
(* PO3 Setpoint Acceleration *)
F_Memcpy(ADR(stControl) + 4, pControlData + 4, 2, stConfig.bSwapProcessData);
(* PO4 Setpoint Deceleration *)
F_Memcpy(ADR(stControl) + 6, pControlData + 6, 2, stConfig.bSwapProcessData);
(* PO5 Digital Outputs *)
F_Memcpy(ADR(stControl) + 8, pControlData + 8, 2, stConfig.bSwapProcessData);
(* PO6 Target Application Mode *)
F_Memcpy(ADR(stControl) + 10, pControlData + 10, 2, stConfig.bSwapProcessData);
(* PO7,PO8 Target Position *)
F_Memcpy(ADR(stControl) + 12, pControlData + 12, 4, stConfig.bSwapProcessData);
END_METHOD

METHOD INTERNAL InitRun
VAR_INST
	bInitRun : BOOL := TRUE;
END_VAR
IF NOT bInitRun THEN RETURN; END_IF
bInitRun := FALSE;

IF pControlData = 0 OR pStatusData = 0 THEN
	ADSLOGSTR(ADSLOG_MSGTYPE_WARN, CONCAT(sPath, ': %s'), 'Plc address not set.');
END_IF

pMovisafe := stConfig.pMovisafeCSSx1a;
fbBasicDrive.fPosition := stConfig.fInitPosition;
END_METHOD

METHOD INTERNAL Operation
VAR_INST
	fTargetPos			: REAL;
	fSetpointVel		: REAL;
	fSetpointAcc		: REAL;
	fSetpointDec		: REAL;
END_VAR
(* Copy setpoint values *)
fTargetPos 		:= DINT_TO_REAL(stControl.nTargetPosition);
fSetpointVel 	:= stControl.nSetpointSpeed * stConfig.fRatioVelocity; 
fSetpointAcc 	:= stControl.nSetpointAcceleration * stConfig.fRatioAccDec;
fSetpointDec 	:= stControl.nSetpointDeceleration * stConfig.fRatioAccDec;

(* Operation statemachine *)
CASE stStatus.nActualApplicationMode OF	
	E_MoviCPositionOperationMode.Jog:
		IF stControl.b4_JoggingCW AND NOT stControl.b5_JoggingCCW THEN
			fbBasicDrive.MoveAbsolute(DINT_TO_REAL(stConfig.nSoftwareLimitMax), fSetpointVel, fSetpointAcc, fSetpointDec);
		ELSIF stControl.b5_JoggingCCW AND NOT stControl.b4_JoggingCW THEN
			fbBasicDrive.MoveAbsolute(DINT_TO_REAL(stConfig.nSoftwareLimitMin), fSetpointVel, fSetpointAcc, fSetpointDec);
		ELSE
			fbBasicDrive.Stop(fSetpointDec);
		END_IF
		
	E_MoviCPositionOperationMode.JogNoEnc:			
		IF stControl.b4_JoggingCW AND NOT stControl.b5_JoggingCCW THEN
			fbBasicDrive.MoveVelocity(fSetpointVel, fSetpointAcc, fSetpointDec);
		ELSIF stControl.b5_JoggingCCW AND NOT stControl.b4_JoggingCW THEN
			fbBasicDrive.MoveVelocity(-fSetpointVel, fSetpointAcc, fSetpointDec);
		ELSE
			fbBasicDrive.Stop(fSetpointDec);
		END_IF
		
	E_MoviCPositionOperationMode.SpeedControl:
		fbBasicDrive.MoveVelocity(fSetpointVel, fSetpointAcc, fSetpointDec);
	
	E_MoviCPositionOperationMode.ReferenceParam:
		//not yet implemented
		
	E_MoviCPositionOperationMode.ReferenceBus:
		//not yet implemented
	
	E_MoviCPositionOperationMode.PositionAbs, E_MoviCPositionOperationMode.EnergyOptimized, E_MoviCPositionOperationMode.MechanicsOptimized:
		IF stControl.b7_StartStop THEN						
			fbBasicDrive.MoveAbsolute(fTargetPos, fSetpointVel, fSetpointAcc, fSetpointDec);
		ELSE
			fbBasicDrive.Stop(fSetpointDec);
		END_IF
	
	E_MoviCPositionOperationMode.PositionRel:
		//not yet implemented
		
	E_MoviCPositionOperationMode.PositionModPos:
		//not yet implemented
		
	E_MoviCPositionOperationMode.PositionModNeg:
		//not yet implemented
		
	E_MoviCPositionOperationMode.PositionModShort:
		//not yet implemented
END_CASE
END_METHOD

METHOD INTERNAL Safety
VAR_INPUT
END_VAR
(* Check if Movisafe is available *)
IF pMovisafe = 0 THEN
	bSTO := TRUE;
	RETURN;
END_IF

(* Safe stop (STO) *)
bSTO := pMovisafe^.stControl.bSTO;
END_METHOD

METHOD INTERNAL SetStatusData
IF pStatusData <= 0 THEN RETURN; END_IF

(* PI1 Status Word *)
F_Memcpy(pStatusData, ADR(stStatus), 2, stConfig.bSwapProcessData);
(* PI2 Actual Speed *)
F_Memcpy(pStatusData + 2, ADR(stStatus) + 2, 2, stConfig.bSwapProcessData);
(* PI3 Actual Status *)
F_Memcpy(pStatusData + 4, ADR(stStatus) + 4, 2, stConfig.bSwapProcessData);
(* PI4 Actual Torque *)
F_Memcpy(pStatusData + 6, ADR(stStatus) + 6, 2, stConfig.bSwapProcessData);
(* PI5 Digital Inputs *)
F_Memcpy(pStatusData + 8, ADR(stStatus) + 8, 2, stConfig.bSwapProcessData);
(* PI6 Actual Application Mode *)
F_Memcpy(pStatusData + 10, ADR(stStatus) + 10, 2, stConfig.bSwapProcessData);
(* PI7,PI8 Actual Position *)
F_Memcpy(pStatusData + 12, ADR(stStatus) + 12, 4, stConfig.bSwapProcessData);
END_METHOD

END_FUNCTION_BLOCK

// Devices/Drives/ProfidriveGSM/FB_ProfidriveGSM
// Profidrive General State Machine
FUNCTION_BLOCK INTERNAL FB_ProfidriveGSM
VAR_INPUT
	bPowerOn					: BOOL := TRUE;
	bStandstill					: BOOL;
	stSTW1 						: ST_ProfiidriveGSM_STW1;
END_VAR

VAR_OUTPUT
	stZSW1						: ST_ProfiidriveGSM_ZSW1;
END_VAR

VAR	
	_eState 					: E_ProfidriveGSM_State := E_ProfidriveGSM_State.S1_SwitchingOnInhibited;	
	rTrig_QuickStop 			: R_TRIG;
	rTrig_Reset 				: R_TRIG;
END_VAR

CASE _eState OF 
	E_ProfidriveGSM_State.S0_Disabled : S0_Disabled();
	E_ProfidriveGSM_State.S1_SwitchingOnInhibited : S1_SwitchingOnInhibited();
	E_ProfidriveGSM_State.S2_ReadyForSwitchingOn : S2_ReadyForSwitchingOn();
	E_ProfidriveGSM_State.S3_SwitchedOn : S3_SwitchedOn();
	E_ProfidriveGSM_State.S4_Operation : S4_Operation();
	E_ProfidriveGSM_State.S51_RampStop : S51_RampStop();
	E_ProfidriveGSM_State.S52_QuickStop : S52_QuickStop();
END_CASE

PROPERTY eState : E_ProfidriveGSM_State
GET
eState := _eState;
END_GET
SET
_eState := eState;
END_SET
END_PROPERTY

PROPERTY PUBLIC nControl : WORD
GET
MEMCPY(ADR(nControl), ADR(stSTW1), 2);
END_GET
SET
MEMCPY(ADR(stSTW1), ADR(nControl), 2);
END_SET
END_PROPERTY

PROPERTY PUBLIC nStatus : WORD
GET
MEMCPY(ADR(nStatus), ADR(stZSW1), 2);
END_GET
SET
MEMCPY(ADR(stZSW1), ADR(nStatus), 2);
END_SET
END_PROPERTY

{ attribute 'hide' }
METHOD PROTECTED S0_Disabled
stZSW1.b0_ReadyToSwitchOn 			:= FALSE;				
stZSW1.b1_ReadyForOperation 		:= FALSE;				
stZSW1.b2_OperationEnabled 			:= FALSE;					
stZSW1.b3_FaultPresent 				:= FALSE;						
stZSW1.b4_CoastStop 				:= FALSE;	 					
stZSW1.b5_QuickStop 				:= FALSE;						
stZSW1.b6_SwitchingOnInhibited 		:= FALSE;				
stZSW1.b7_WarningPresent			:= FALSE;			
stZSW1.b9_ControlRequested 			:= FALSE;	

(*to S1*)	
IF bPowerOn THEN
	_eState := E_ProfidriveGSM_State.S1_SwitchingOnInhibited;
END_IF
END_METHOD

{ attribute 'hide' }
METHOD INTERNAL S1_SwitchingOnInhibited
VAR_INPUT
END_VAR
stZSW1.b0_ReadyToSwitchOn 		:= FALSE;				
stZSW1.b1_ReadyForOperation 		:= FALSE;				
stZSW1.b2_OperationEnabled 		:= FALSE;						
stZSW1.b6_SwitchingOnInhibited 	:= TRUE;

(*to S2_ReadyForSwitchingOn*)	
IF NOT stSTW1.b0_On AND stSTW1.b1_CoastStop AND stSTW1.b2_QuickStop THEN
	_eState := E_ProfidriveGSM_State.S2_ReadyForSwitchingOn;
END_IF
END_METHOD

{ attribute 'hide' }
METHOD INTERNAL S2_ReadyForSwitchingOn
VAR_INPUT
END_VAR
stZSW1.b0_ReadyToSwitchOn 		:= TRUE;				
stZSW1.b1_ReadyForOperation 		:= FALSE;				
stZSW1.b2_OperationEnabled 		:= FALSE;						
stZSW1.b6_SwitchingOnInhibited 	:= FALSE;

(*to S1_SwitchingOnInhibited*)	
IF NOT stSTW1.b1_CoastStop OR NOT stSTW1.b2_QuickStop THEN
	_eState := E_ProfidriveGSM_State.S1_SwitchingOnInhibited;
	RETURN;
END_IF

(*to S3_SwitchedOn*)	
IF stSTW1.b0_On THEN
	_eState := E_ProfidriveGSM_State.S3_SwitchedOn;
END_IF
END_METHOD

{ attribute 'hide' }
METHOD INTERNAL S3_SwitchedOn
VAR_INPUT
END_VAR
stZSW1.b0_ReadyToSwitchOn 		:= TRUE;				
stZSW1.b1_ReadyForOperation 		:= TRUE;				
stZSW1.b2_OperationEnabled 		:= FALSE;						
stZSW1.b6_SwitchingOnInhibited 	:= FALSE;

(*to S1_SwitchingOnInhibited*)	
IF NOT stSTW1.b1_CoastStop OR NOT stSTW1.b2_QuickStop THEN
	_eState := E_ProfidriveGSM_State.S1_SwitchingOnInhibited;
	RETURN;
END_IF

(*to S2_ReadyForSwitchingOn*)	
IF NOT stSTW1.b0_On THEN
	_eState := E_ProfidriveGSM_State.S2_ReadyForSwitchingOn;
	RETURN;
END_IF

(*to S4_Operation*)	
IF stSTW1.b3_EnableOperation THEN
	_eState := E_ProfidriveGSM_State.S4_Operation;
END_IF
END_METHOD

{ attribute 'hide' }
METHOD INTERNAL S4_Operation
VAR_INPUT
END_VAR
stZSW1.b0_ReadyToSwitchOn 		:= TRUE;				
stZSW1.b1_ReadyForOperation 		:= TRUE;				
stZSW1.b2_OperationEnabled 		:= TRUE;					
stZSW1.b6_SwitchingOnInhibited 	:= FALSE;

(*to S1_SwitchingOnInhibited*)	
IF NOT stSTW1.b1_CoastStop THEN
	_eState := E_ProfidriveGSM_State.S1_SwitchingOnInhibited;
	RETURN;
END_IF

(*to S52_QuickStop*)	
IF NOT stSTW1.b2_QuickStop THEN
	_eState := E_ProfidriveGSM_State.S52_QuickStop;
	RETURN;
END_IF

(*to S51_RampStop*)	
IF NOT stSTW1.b0_On THEN
	_eState := E_ProfidriveGSM_State.S51_RampStop;
	RETURN;
END_IF

(*to S3_SwitchedOn*)	
IF NOT stSTW1.b3_EnableOperation THEN
	_eState := E_ProfidriveGSM_State.S3_SwitchedOn;
END_IF
END_METHOD

{ attribute 'hide' }
METHOD INTERNAL S51_RampStop
VAR_INPUT
END_VAR
stZSW1.b0_ReadyToSwitchOn 		:= TRUE;				
stZSW1.b1_ReadyForOperation 		:= TRUE;				
stZSW1.b2_OperationEnabled 		:= FALSE;					
stZSW1.b6_SwitchingOnInhibited 	:= FALSE;

(*to S1_SwitchingOnInhibited*)	
IF NOT stSTW1.b1_CoastStop THEN
	_eState := E_ProfidriveGSM_State.S1_SwitchingOnInhibited;
	RETURN;
END_IF

(*to S52_QuickStop*)	
IF NOT stSTW1.b2_QuickStop THEN
	_eState := E_ProfidriveGSM_State.S52_QuickStop;
	RETURN;
END_IF

(*to S2_ReadyForSwitchingOn*)	
IF NOT stSTW1.b3_EnableOperation OR bStandstill THEN
	_eState := E_ProfidriveGSM_State.S2_ReadyForSwitchingOn;
END_IF

(*to S4_Operation*)	
IF stSTW1.b0_On THEN
	_eState := E_ProfidriveGSM_State.S4_Operation;
	RETURN;
END_IF
END_METHOD

{ attribute 'hide' }
METHOD INTERNAL S52_QuickStop
VAR_INPUT
END_VAR
stZSW1.b0_ReadyToSwitchOn 		:= TRUE;				
stZSW1.b1_ReadyForOperation 		:= TRUE;				
stZSW1.b2_OperationEnabled 		:= FALSE;					
stZSW1.b6_SwitchingOnInhibited 	:= FALSE;

(*to S1_SwitchingOnInhibited*)	
IF NOT stSTW1.b1_CoastStop THEN
	_eState := E_ProfidriveGSM_State.S1_SwitchingOnInhibited;
	RETURN;
END_IF

(*to S1_SwitchingOnInhibited*)	
IF NOT stSTW1.b3_EnableOperation OR bStandstill THEN
	_eState := E_ProfidriveGSM_State.S1_SwitchingOnInhibited;
END_IF
END_METHOD

END_FUNCTION_BLOCK

// Devices/Drives/MovisafeCSSx1a/FB_MovisafeCSSx1a
{attribute 'reflection'}
FUNCTION_BLOCK FB_MovisafeCSSx1a EXTENDS FB_Base
VAR_INPUT
	bASF_DIAG			: BOOL; //At least one drive safety function has exceeded a limit
	bSBT_ACTIVE 		: BOOL; //Brake test is active
	bF_DI0				: BOOL; //State digital input 1
	bF_DI1				: BOOL; //State digital input 2
	bF_DI2				: BOOL; //State digital input 3
	bF_DI3				: BOOL; //State digital input 4
	bSSM_1				: BOOL; //SSM 1 ist activated (Safe speed monitoring)
	bSSM_2				: BOOL; //SSM 2 ist activated (Safe speed monitoring)
	bSSM_3				: BOOL;	//SSM 3 ist activated (Safe speed monitoring)
	bSSM_4				: BOOL; //SSM 4 ist activated (Safe speed monitoring)
	stControl			: ST_MovisafeCSSx1a_Control;
	stConfig			: ST_MovisafeCSSx1a_Config;
END_VAR

VAR_OUTPUT	
	stStatus			: ST_MovisafeCSSx1a_Status;
END_VAR

VAR
    {attribute 'instance-path'} 
    {attribute 'noinit'} 
    sPath 				: STRING; 
	pControlData		: POINTER TO BYTE;
	pStatusData			: POINTER TO BYTE;
END_VAR

SUPER^();
InitRun();

GetControlData();
ControlLogic();
SetStatusData();

(*Assign Process Data Objects to device*)
METHOD PUBLIC AssignProcessData : BOOL
VAR_INPUT
	aControlData 		: ANY; //Addr. Process Output
	aStatusData 		: ANY; //Addr. Process Input
END_VAR
THIS^.pControlData := aControlData.pValue;
THIS^.pStatusData := aStatusData.pValue;
END_METHOD

METHOD INTERNAL ControlLogic : BOOL
VAR_INPUT
END_VAR
stStatus.bSTO_ACTIVE		:= stControl.bSTO;
stStatus.bASF_DIAG			:= bASF_DIAG;
stStatus.bSBT_ACTIVE		:= bSBT_ACTIVE;
stStatus.bINPUT_DATA_VALID	:= TRUE;
stStatus.bMUTING_ENC_ERR	:= stControl.bMUTING_ENC_ERR;
stStatus.bTEST_MODE_ACTIVE	:= stControl.bTEST_MODE_ACTIVE;
stStatus.bWARNING			:= FALSE;
stStatus.bERROR_STATE		:= FALSE;
stStatus.bF_DI0				:= bF_DI0;
stStatus.bF_DI1				:= bF_DI1;
stStatus.bF_DI2				:= bF_DI2;
stStatus.bF_DI3				:= bF_DI3;
stStatus.bRES_14			:= FALSE;
stStatus.bRES_15			:= FALSE;
stStatus.bRES_16			:= FALSE;
stStatus.bRES_17			:= FALSE;
stStatus.bSOS_1				:= NOT stControl.bSOS_1;
stStatus.bRES_21			:= FALSE;
stStatus.bSSx1				:= NOT stControl.bSSx1;
stStatus.bSSx2				:= NOT stControl.bSSx2;
stStatus.bSDI_1				:= NOT stControl.bSDI_1;
stStatus.bSDI_2				:= NOT stControl.bSDI_2;
stStatus.bSLI_1				:= NOT stControl.bSLI_1;
stStatus.bSLI_2				:= NOT stControl.bSLI_1;
stStatus.bSLS_1				:= NOT stControl.bSLS_1;
stStatus.bSLS_2				:= NOT stControl.bSLS_2;
stStatus.bSLS_3				:= NOT stControl.bSLS_3;
stStatus.bSLS_4				:= NOT stControl.bSLS_4;
stStatus.bSSR_1				:= NOT stControl.bSSR_1;
stStatus.bSSR_2				:= NOT stControl.bSSR_2;
stStatus.bRES_36			:= FALSE;
stStatus.bRES_37			:= FALSE;
stStatus.bSLA_1				:= NOT stControl.bSLA_1;
stStatus.bSLA_2				:= NOT stControl.bSLA_2;
stStatus.bSSM_1				:= bSSM_1;
stStatus.bSSM_2				:= bSSM_2;
stStatus.bSSM_3				:= bSSM_3;
stStatus.bSSM_4				:= bSSM_4;
stStatus.bRES_46			:= FALSE;
stStatus.bRES_47			:= FALSE;
stStatus.bRES_50			:= FALSE;
stStatus.bRES_51			:= FALSE;
stStatus.bRES_52			:= FALSE;
stStatus.bRES_53			:= FALSE;
stStatus.bRES_54			:= FALSE;
stStatus.bRES_55			:= FALSE;
stStatus.bRES_56			:= FALSE;
stStatus.bRES_57			:= FALSE;
END_METHOD

METHOD INTERNAL GetControlData
VAR_INPUT
END_VAR
IF pControlData <= 0 THEN RETURN; END_IF

F_MEMCPY(ADR(stControl), pControlData, 5, stConfig.bSwapProcessData);
END_METHOD

METHOD INTERNAL InitRun
VAR_INST
	bInitRun : BOOL := TRUE;
END_VAR
IF NOT bInitRun THEN RETURN; END_IF
bInitRun := FALSE;

IF pControlData = 0 OR pStatusData = 0 THEN
	ADSLOGSTR(ADSLOG_MSGTYPE_WARN, CONCAT(sPath, ': %s'), 'Plc address not set.');
END_IF
END_METHOD

METHOD INTERNAL SetStatusData
VAR_INPUT
END_VAR
IF pStatusData <= 0 THEN RETURN; END_IF

F_MEMCPY(pStatusData, ADR(stStatus), 6, stConfig.bSwapProcessData);
END_METHOD

END_FUNCTION_BLOCK

// Devices/Drives/MoviCVelocity/FB_MoviCVelocity
{attribute 'reflection'}
FUNCTION_BLOCK FB_MoviCVelocity EXTENDS FB_LinkDataReal
VAR_INPUT
	bSTO						: BOOL := TRUE;
	stControl 					: ST_MoviCVelocity_Control;
	stConfig					: ST_MoviCVelocity_Config;
END_VAR

VAR_OUTPUT
	stStatus					: ST_MoviCVelocity_Status;
	fValue						: REAL;
END_VAR

VAR
    {attribute 'instance-path'} 
    {attribute 'noinit'} 
    sPath 						: STRING; 	                			
	                			
	fbBaseState					: FB_ProfidriveGSM;
	fbBasicDrive				: FB_DriveControl;	                				
	
	pMovisafe					: POINTER TO FB_MovisafeCSSx1a;		
	pControlData				: POINTER TO BYTE; //Addr. Process Output
	pStatusData					: POINTER TO BYTE; //Addr. Process Input
END_VAR

SUPER^();
InitRun();

GetControlData();
Safety();
ControlLogic();
SetStatusData();

(*Assign Process Data Objects to device*)
METHOD PUBLIC AssignProcessData : BOOL
VAR_INPUT
	aControlData 		: ANY; //Addr. Process Output
	aStatusData 		: ANY; //Addr. Process Input
END_VAR
THIS^.pControlData := aControlData.pValue;
THIS^.pStatusData := aStatusData.pValue;
END_METHOD

METHOD INTERNAL ControlLogic
(* Base state of the controller *)
fbBaseState.bStandstill := OC_Core.F_Compare(fbBasicDrive.fVelocity, 0, 1E-3);
fbBaseState.stSTW1.b0_On := stControl.b1_EnableBusStop AND fbBaseState.eState <> E_ProfidriveGSM_State.S1_SwitchingOnInhibited;
fbBaseState.stSTW1.b1_CoastStop := NOT stControl.b13_ActivateInhibit AND bSTO;
fbBaseState.stSTW1.b2_QuickStop := stControl.b0_EnableEStop;
fbBaseState.stSTW1.b3_EnableOperation := stControl.b7_StartStop;

fbBaseState();
					
(* Evaluate base state *)
CASE fbBaseState.eState OF	
(* S1, S2 or S3 -> Drive coasts to a stop or brake is applied *)
	E_ProfidriveGSM_State.S1_SwitchingOnInhibited,
	E_ProfidriveGSM_State.S2_ReadyForSwitchingOn,
	E_ProfidriveGSM_State.S3_SwitchedOn:
		fbBasicDrive.Stop(stConfig.fDecCoastStop);

(* S4 -> Operation mode *)
	E_ProfidriveGSM_State.S4_Operation:
		Operation();

(* S5a -> Drive decelerates with application limit *)
	E_ProfidriveGSM_State.S51_RampStop:
		fbBasicDrive.Stop(stConfig.fDecelerationLimit);
		
(* S5b -> Drive decelerates with emergency stop ramp *)
	E_ProfidriveGSM_State.S52_QuickStop:
	    fbBasicDrive.Stop(stConfig.fDecEstop);
END_CASE
	
(* Status Word *)
stStatus.b0_InverterReady				:= TRUE;
stStatus.b1_STOInactive					:= bSTO;
stStatus.b2_PowerStageOn				:= fbBaseState.bPowerOn;
stStatus.b3_BrakeReleased				:= stControl.b1_EnableBusStop OR stControl.b3_ReleaseBrake;
stStatus.b4_MotorTurning				:= NOT fbBaseState.bStandstill;
stStatus.b5_DriveReferenced				:= TRUE;
stStatus.b6_SetpointsActive		 		:= FALSE;
stStatus.b7_TargetpositionReached		:= FALSE;	
stStatus.b8_ErrorActive					:= FALSE;
stStatus.b9_WarningActive				:= FALSE;
stStatus.b10_DriveTrain2Active			:= stControl.b10_ActivateDriveTrain2;
stStatus.b11_SpeedSetpointReached		:= fbBasicDrive.bIsMoving;
stStatus.b12_SoftwareLimitsDisabled		:= stControl.b12_DisableSoftwareLimits;
stStatus.b13_OutputStageInhibit			:= fbBaseState.stZSW1.b6_SwitchingOnInhibited;
stStatus.b14_StandByModeActive			:= stControl.b14_ActivateStandByMode;
stStatus.b15_MovikitHeartbeat			:= stControl.b15_MovikitHeartbeat;

(* Status values *)
stStatus.nActualSpeed := REAL_TO_INT(fbBasicDrive.fVelocity / stConfig.fRatioVelocity);
stStatus.nActualStatus := 0;
stStatus.nActualTorque := 0;
stStatus.nDigitalInputs := 0;
	
(* Output of actual value *)	
IF stConfig.bOutputVelocity THEN
	ControlData := fbBasicDrive.fVelocity / stConfig.fRatioVelocity;
ELSE
	ControlData := ControlData + fbBasicDrive.fVelocity / stConfig.fRatioVelocity *  GVL_Core.fbSystem.fDeltaTime * GVL_Core.fbSystem.fTimeScaling;
END_IF

fValue := ControlData;
END_METHOD

METHOD INTERNAL GetControlData : BOOL
IF pControlData <= 0 THEN RETURN; END_IF

(* PO1 Control Word *)
F_Memcpy(ADR(stControl), pControlData, 2, stConfig.bSwapProcessData);
(* PO2 Setpoint Speed *)
F_Memcpy(ADR(stControl) + 2, pControlData + 2, 2, stConfig.bSwapProcessData);
(* PO3 Setpoint Acceleration *)
F_Memcpy(ADR(stControl) + 4, pControlData + 4, 2, stConfig.bSwapProcessData);
(* PO4 Setpoint Deceleration *)
F_Memcpy(ADR(stControl) + 6, pControlData + 6, 2, stConfig.bSwapProcessData);
(* PO5 Digital Outputs *)
F_Memcpy(ADR(stControl) + 8, pControlData + 8, 2, stConfig.bSwapProcessData);
END_METHOD

METHOD INTERNAL InitRun
VAR_INST
	bInitRun : BOOL := TRUE;
END_VAR
IF NOT bInitRun THEN RETURN; END_IF
bInitRun := FALSE;

IF pControlData = 0 OR pStatusData = 0 THEN
	ADSLOGSTR(ADSLOG_MSGTYPE_WARN, CONCAT(sPath, ': %s'), 'Plc address not set.');
END_IF

pMovisafe := stConfig.pMovisafeCSSx1a;
fbBasicDrive.fPosition := stConfig.fInitPosition;
END_METHOD

METHOD INTERNAL Operation
VAR_INST
	fTargetPos			: REAL;
	fSetpointVel		: REAL;
	fSetpointAcc		: REAL;
	fSetpointDec		: REAL;
END_VAR
(* Copy setpoint values *)
fSetpointVel 	:= stControl.nSetpointSpeed * stConfig.fRatioVelocity; 
fSetpointAcc 	:= stControl.nSetpointAcceleration * stConfig.fRatioAccDec;

fbBasicDrive.MoveVelocity(fSetpointVel, fSetpointAcc, fSetpointAcc);
END_METHOD

METHOD INTERNAL Safety
VAR_INPUT
END_VAR
(* Check if Movisafe is available *)
IF pMovisafe = 0 THEN
	bSTO := TRUE;
	RETURN;
END_IF

(* Safe stop (STO) *)
bSTO := pMovisafe^.stControl.bSTO;
END_METHOD

METHOD INTERNAL SetStatusData
IF pStatusData <= 0 THEN RETURN; END_IF

(* PI1 Status Word *)
F_Memcpy(pStatusData, ADR(stStatus), 2, stConfig.bSwapProcessData);
(* PI2 Actual Speed *)
F_Memcpy(pStatusData + 2, ADR(stStatus) + 2, 2, stConfig.bSwapProcessData);
(* PI3 Actual Status *)
F_Memcpy(pStatusData + 4, ADR(stStatus) + 4, 2, stConfig.bSwapProcessData);
(* PI4 Actual Torque *)
F_Memcpy(pStatusData + 6, ADR(stStatus) + 6, 2, stConfig.bSwapProcessData);
(* PI5 Digital Inputs *)
F_Memcpy(pStatusData + 8, ADR(stStatus) + 8, 2, stConfig.bSwapProcessData);
END_METHOD

END_FUNCTION_BLOCK

// Devices/Drives/MovisafeCSBx1a/FB_MovisafeCSBx1a
{attribute 'reflection'}
FUNCTION_BLOCK FB_MovisafeCSBx1a EXTENDS FB_DeviceByte
VAR_INPUT	
	bF_DI0				: BOOL; //State digital input 1
	bF_DI1				: BOOL; //State digital input 2
	bF_DI2				: BOOL; //State digital input 3
	bF_DI3				: BOOL; //State digital input 4
	stControl			: ST_MovisafeCSBx1a_Control;
	stConfig 			: ST_MovisafeCSBx1a_Config;
END_VAR

VAR_OUTPUT	
	stStatus			: ST_MovisafeCSBx1a_Status;
END_VAR

VAR
    {attribute 'instance-path'} 
    {attribute 'noinit'} 
    sPath 				: STRING; 
	pControlData		: POINTER TO BYTE;
	pStatusData			: POINTER TO BYTE;
END_VAR

SUPER^();
InitRun();

GetControlData();
ControlLogic();
SetStatusData();

(*Assign Process Data Objects to device*)
METHOD PUBLIC AssignProcessData : BOOL
VAR_INPUT
	aControlData 		: ANY; //Addr. Process Output 3 Bytes
	aStatusData 		: ANY; //Addr. Process Input 4 Bytes
END_VAR
THIS^.pControlData := aControlData.pValue;
THIS^.pStatusData := aStatusData.pValue;
END_METHOD

METHOD INTERNAL ControlLogic : BOOL
VAR_INPUT
END_VAR
stStatus.b0_STO_ACTIVE			:= NOT stControl.b0_STO1;
stStatus.b3_INPUT_DATA_VALID	:= TRUE;
stStatus.b6_WARNING				:= FALSE;
stStatus.b7_ERROR_STATE			:= FALSE;
stStatus.b8_F_DI0				:= bF_DI0;
stStatus.b9_F_DI1				:= bF_DI1;
stStatus.b10_F_DI2				:= bF_DI2;
stStatus.b11_F_DI3				:= bF_DI3;
stStatus.b18_SSx1				:= stControl.b18_SSx1;
stStatus.b19_SSx2				:= stControl.b19_SSx2;
END_METHOD

METHOD INTERNAL GetControlData
VAR_INPUT
END_VAR
IF pControlData <= 0 THEN RETURN; END_IF

F_MEMCPY(ADR(stControl), pControlData, 3, stConfig.bSwapProcessData);
END_METHOD

METHOD INTERNAL InitRun
VAR_INST
	bInitRun : BOOL := TRUE;
END_VAR
IF NOT bInitRun THEN RETURN; END_IF
bInitRun := FALSE;

IF pControlData = 0 OR pStatusData = 0 THEN
	ADSLOGSTR(ADSLOG_MSGTYPE_WARN, CONCAT(sPath, ': %s'), 'Plc address not set.');
END_IF
END_METHOD

METHOD INTERNAL SetStatusData
VAR_INPUT
END_VAR
IF pStatusData <= 0 THEN RETURN; END_IF

F_MEMCPY(pStatusData, ADR(stStatus), 4, stConfig.bSwapProcessData);
END_METHOD

END_FUNCTION_BLOCK

// Devices/Drives/ProfidriveTelegram1/FB_ProfidriveTelegram1
{attribute 'reflection'} 
FUNCTION_BLOCK FB_ProfidriveTelegram1 EXTENDS FB_LinkDataReal
VAR_INPUT	
	stControl					: ST_ProfidriveTelegram1_Control;
	stConfig 					: ST_ProfidriveTelegram1_Config;
END_VAR

VAR_OUTPUT
	stStatus					: ST_ProfidriveTelegram1_Status;
	fValue						: REAL;
END_VAR

VAR
    {attribute 'instance-path'} 
    {attribute 'noinit'} 
    sPath 						: STRING; 	
	                        	
	fbProfidriveGSM				: FB_ProfidriveGSM;	
	fbMoveVelocity				: FB_MoveVelocity;
	                        	
	fAcceleration	 			: REAL;
	fDeceleration		 		: REAL;
	fDecelerationQuickStop 		: REAL;
	fDecelerationCoastStop 		: REAL;
	bQuickStopExternal			: BOOL;
	
	pControlData				: POINTER TO BYTE; //Addr. Process Output, 4 BYTES FROM FIELDBUS
	pStatusData					: POINTER TO BYTE; //Addr. Process Input, 4 BYTES TO FIELDBUS
END_VAR

SUPER^();
InitRun();

GetControlData();
ControlLogic();
SetStatusData();

(*Assign Process Data Objects to device*)
METHOD PUBLIC AssignProcessData : BOOL
VAR_INPUT
	aControlData 		: ANY; //Addr. Process Output, 4 BYTES FROM FIELDBUS
	aStatusData 		: ANY; //Addr. Process Input, 4 BYTES TO FIELDBUS
END_VAR
THIS^.pControlData := aControlData.pValue;
THIS^.pStatusData := aStatusData.pValue;
END_METHOD

METHOD INTERNAL ControlLogic
(*Initialize Init Value*)
IF SUPER^.Status.7 THEN
	ControlData := StatusData;
END_IF

(* Call base statemachine *)
fbProfidriveGSM.bStandstill						:= OC_Core.F_Compare(fbMoveVelocity.fVelocity, 0, 1E-3);
fbProfidriveGSM.stSTW1.b0_On 					:= stControl.b0_OFF1;
fbProfidriveGSM.stSTW1.b1_CoastStop 			:= stControl.b1_OFF2;
fbProfidriveGSM.stSTW1.b2_QuickStop 			:= stControl.b2_OFF3 AND NOT bQuickStopExternal;
fbProfidriveGSM.stSTW1.b3_EnableOperation		:= stControl.b3_EnableOperation;

(* Preset target values *)
fbMoveVelocity.fTargetVelocity					:= 0;
fbMoveVelocity.fAccMax 							:= fAcceleration;
fbMoveVelocity.fDecMax 							:= fDeceleration;

(* Operation Logic *)
Operation();
	
(* Coast stop, Quick stop, Ramp stop *)
IF fbProfidriveGSM.eState = E_ProfidriveGSM_State.S1_SwitchingOnInhibited THEN
	fbMoveVelocity.fTargetVelocity := 0;
	fbMoveVelocity.fAccMax := fDecelerationCoastStop;
	fbMoveVelocity.fDecMax := fDecelerationCoastStop;
ELSIF fbProfidriveGSM.eState = E_ProfidriveGSM_State.S52_QuickStop THEN
	fbMoveVelocity.fTargetVelocity := 0;
	fbMoveVelocity.fAccMax := fDecelerationQuickStop;
	fbMoveVelocity.fDecMax := fDecelerationQuickStop;
ELSIF fbProfidriveGSM.eState = E_ProfidriveGSM_State.S51_RampStop THEN
	fbMoveVelocity.fTargetVelocity := 0;
	fbMoveVelocity.fAccMax := fDeceleration;
	fbMoveVelocity.fDecMax := fDeceleration;
END_IF

(* Call MoveVelocity *)
fbMoveVelocity();
	
(* Status word *)
stStatus.b0_ReadyForSwitchingOn				:= fbProfidriveGSM.stZSW1.b0_ReadyToSwitchOn;	
stStatus.b1_ReadyForOperation				:= fbProfidriveGSM.stZSW1.b1_ReadyForOperation;
stStatus.b2_OperationEnabled				:= stControl.b3_EnableOperation;
stStatus.b3_FaultPresent					:= FALSE;
stStatus.b4_NoCoastDownActive				:= fbProfidriveGSM.eState <> E_ProfidriveGSM_State.S1_SwitchingOnInhibited;
stStatus.b5_NoQuickStopActive				:= fbProfidriveGSM.eState <> E_ProfidriveGSM_State.S52_QuickStop;
stStatus.b6_SwitchingOnInhibited			:= fbProfidriveGSM.stZSW1.b6_SwitchingOnInhibited;
stStatus.b7_AlarmPresent					:= FALSE;
stStatus.b8_DeviationWithinTolerance		:= TRUE;
stStatus.b9_ControlRequested				:= stConfig.bControlRequested;
stStatus.b10_RpmCompValueReachedOrExceeded	:= fbMoveVelocity.bIsReached;
stStatus.b11_TorqueOrPowerLimitNotReached	:= TRUE;
stStatus.b12_OpenHoldingBrake 				:= fbProfidriveGSM.eState > E_ProfidriveGSM_State.S3_SwitchedOn;
stStatus.b13_NoOvertempAlarm				:= TRUE;	
stStatus.b14_MotorRotatesForwards			:= fbMoveVelocity.fVelocity >= 0;
stStatus.b15_NoAlarmNoOvertempPowerUnit		:= TRUE;

(* Reset quickstop from extern *)
IF stControl.b7_AcknowledgeFaults THEN
	bQuickStopExternal := FALSE;
END_IF

(* Calculate NIST *)
IF stConfig.fP2000 = 0 THEN
	stStatus.nNIst	:= 0;
ELSE
	stStatus.nNIst	:=	REAL_TO_INT((fbMoveVelocity.fVelocity * 16#4000) / stConfig.fP2000);
END_IF

(* Output of actual value *)	
IF stConfig.bOutputVelocity THEN
	ControlData := fbMoveVelocity.fVelocity;
ELSE
	ControlData := ControlData + fbMoveVelocity.fVelocity *  GVL_Core.fbSystem.fDeltaTime * GVL_Core.fbSystem.fTimeScaling;
END_IF

fValue := ControlData;
END_METHOD

METHOD INTERNAL GetControlData : BOOL
VAR	
	nBufferWord 	: WORD;
END_VAR
IF pControlData <= 0 THEN RETURN; END_IF

F_Memcpy(ADR(stControl), pControlData, 2, stConfig.bSwapProcessData);
F_Memcpy(ADR(stControl) + 2, pControlData + 2, 2, stConfig.bSwapProcessData);
END_METHOD

METHOD INTERNAL InitRun : BOOL
VAR_INST
	bInitRun : BOOL := TRUE;
END_VAR
IF NOT bInitRun THEN RETURN; END_IF
bInitRun := FALSE;

IF pControlData = 0 OR pStatusData = 0 THEN
	ADSLOGSTR(ADSLOG_MSGTYPE_WARN, CONCAT(sPath, ': %s'), 'Plc address not set.');
END_IF
END_METHOD

METHOD PRIVATE Operation : BOOL
IF fbProfidriveGSM.eState = E_ProfidriveGSM_State.S4_Operation THEN	
	// Main setpoint
	IF NOT stControl.b8_Jog1 AND NOT stControl.b9_Jog2 THEN
		fbMoveVelocity.fTargetVelocity := (stControl.nNSoll * stConfig.fP2000) / 16#4000;
	// Jog 1
	ELSIF stControl.b8_Jog1 AND NOT stControl.b9_Jog2 THEN
		fbMoveVelocity.fTargetVelocity := stConfig.fP1058;
	// Jog 2
	ELSIF NOT stControl.b8_Jog1 AND stControl.b9_Jog2 THEN	
		fbMoveVelocity.fTargetVelocity := stConfig.fP1059;
	END_IF
	// Stop
	IF NOT stControl.b4_OperatingCondition OR NOT stControl.b6_EnableSetpoint THEN
		fbMoveVelocity.fTargetVelocity := 0;
	END_IF
	// Invert velocity
	IF stControl.b11_SetpointInversion THEN
		fbMoveVelocity.fTargetVelocity := -fbMoveVelocity.fTargetVelocity;
	END_IF	
	// Hold velocity
	IF NOT stControl.b5_ContinueRampFunctionGenerator AND NOT stControl.b8_Jog1 AND NOT stControl.b9_Jog2 THEN
		fbMoveVelocity.fTargetVelocity := fbMoveVelocity.fVelocity;
	END_IF	
END_IF
END_METHOD

METHOD INTERNAL SetStatusData
IF pStatusData <= 0 THEN RETURN; END_IF

F_Memcpy(pStatusData, ADR(stStatus), 2, stConfig.bSwapProcessData);
F_Memcpy(pStatusData + 2, ADR(stStatus) + 2, 2, stConfig.bSwapProcessData);
END_METHOD

END_FUNCTION_BLOCK

// Tests/Drives/FB_ProfidriveGSM_Test
FUNCTION_BLOCK FB_ProfidriveGSM_Test EXTENDS TcUnit.FB_TestSuite

TestState_S0();
TestState_S1();
TestState_S2();
TestState_S3();
TestState_S4();
TestState_S51();
TestState_S52();

TestTransitions_S0();
TestTransitions_S1();
TestTransitions_S2();
TestTransitions_S3();
TestTransitions_S4();
TestTransitions_S51();
TestTransitions_S52();

METHOD TestState_S0 : BOOL
VAR
	fbFSM 				: FB_ProfidriveGSM;
	stStatusExpected	: ST_ProfiidriveGSM_ZSW1;
	nStatusExpected 	: WORD;
END_VAR
TEST('Set State S0');

//Arrange
fbFSM.eState := E_ProfidriveGSM_State.S0_Disabled;

stStatusExpected.b0_ReadyToSwitchOn 		:= FALSE;				
stStatusExpected.b1_ReadyForOperation 		:= FALSE;				
stStatusExpected.b2_OperationEnabled 		:= FALSE;
stStatusExpected.b6_SwitchingOnInhibited 	:= FALSE;
MEMCPY(ADR(nStatusExpected), ADR(stStatusExpected), 2);

//Act
fbFSM();

//Assert
IF (nStatusExpected <> fbFSM.nStatus) THEN
	AssertEquals_BOOL(stStatusExpected.b0_ReadyToSwitchOn, fbFSM.stZSW1.b0_ReadyToSwitchOn, 'b0_ReadyToSwitchOn: AssertEquals not returning expected value');
	AssertEquals_BOOL(stStatusExpected.b1_ReadyForOperation, fbFSM.stZSW1.b1_ReadyForOperation, 'b1_ReadyForOperation: AssertEquals not returning expected value');
	AssertEquals_BOOL(stStatusExpected.b2_OperationEnabled, fbFSM.stZSW1.b2_OperationEnabled, 'b2_OperationEnabled: AssertEquals not returning expected value');	
	AssertEquals_BOOL(stStatusExpected.b6_SwitchingOnInhibited, fbFSM.stZSW1.b6_SwitchingOnInhibited, 'b6_SwitchingOnInhibited: AssertEquals not returning expected value');	
END_IF

TEST_FINISHED();
END_METHOD

METHOD TestState_S1 : BOOL
VAR
	fbFSM 				: FB_ProfidriveGSM;
	stStatusExpected	: ST_ProfiidriveGSM_ZSW1;
	nStatusExpected 	: WORD;
END_VAR
TEST('Set State S1');

//Arrange
fbFSM.eState := E_ProfidriveGSM_State.S1_SwitchingOnInhibited;

stStatusExpected.b0_ReadyToSwitchOn 		:= FALSE;				
stStatusExpected.b1_ReadyForOperation 		:= FALSE;				
stStatusExpected.b2_OperationEnabled 		:= FALSE;
stStatusExpected.b6_SwitchingOnInhibited 	:= TRUE;
MEMCPY(ADR(nStatusExpected), ADR(stStatusExpected), 2);

//Act
fbFSM();

//Assert
IF (nStatusExpected <> fbFSM.nStatus) THEN
	AssertEquals_BOOL(stStatusExpected.b0_ReadyToSwitchOn, fbFSM.stZSW1.b0_ReadyToSwitchOn, 'b0_ReadyToSwitchOn: AssertEquals not returning expected value');
	AssertEquals_BOOL(stStatusExpected.b1_ReadyForOperation, fbFSM.stZSW1.b1_ReadyForOperation, 'b1_ReadyForOperation: AssertEquals not returning expected value');
	AssertEquals_BOOL(stStatusExpected.b2_OperationEnabled, fbFSM.stZSW1.b2_OperationEnabled, 'b2_OperationEnabled: AssertEquals not returning expected value');	
	AssertEquals_BOOL(stStatusExpected.b6_SwitchingOnInhibited, fbFSM.stZSW1.b6_SwitchingOnInhibited, 'b6_SwitchingOnInhibited: AssertEquals not returning expected value');	
END_IF

TEST_FINISHED();
END_METHOD

METHOD TestState_S2 : BOOL
VAR
	fbFSM 				: FB_ProfidriveGSM;
	stStatusExpected	: ST_ProfiidriveGSM_ZSW1;
	nStatusExpected 	: WORD;
END_VAR
TEST('Set State S2');

//Arrange
fbFSM.eState := E_ProfidriveGSM_State.S2_ReadyForSwitchingOn;

stStatusExpected.b0_ReadyToSwitchOn 		:= TRUE;				
stStatusExpected.b1_ReadyForOperation 		:= FALSE;				
stStatusExpected.b2_OperationEnabled 		:= FALSE;
stStatusExpected.b6_SwitchingOnInhibited 	:= FALSE;
MEMCPY(ADR(nStatusExpected), ADR(stStatusExpected), 2);

//Act
fbFSM();

//Assert
IF (nStatusExpected <> fbFSM.nStatus) THEN
	AssertEquals_BOOL(stStatusExpected.b0_ReadyToSwitchOn, fbFSM.stZSW1.b0_ReadyToSwitchOn, 'b0_ReadyToSwitchOn: AssertEquals not returning expected value');
	AssertEquals_BOOL(stStatusExpected.b1_ReadyForOperation, fbFSM.stZSW1.b1_ReadyForOperation, 'b1_ReadyForOperation: AssertEquals not returning expected value');
	AssertEquals_BOOL(stStatusExpected.b2_OperationEnabled, fbFSM.stZSW1.b2_OperationEnabled, 'b2_OperationEnabled: AssertEquals not returning expected value');	
	AssertEquals_BOOL(stStatusExpected.b6_SwitchingOnInhibited, fbFSM.stZSW1.b6_SwitchingOnInhibited, 'b6_SwitchingOnInhibited: AssertEquals not returning expected value');	
END_IF

TEST_FINISHED();
END_METHOD

METHOD TestState_S3 : BOOL
VAR
	fbFSM 				: FB_ProfidriveGSM;
	stStatusExpected	: ST_ProfiidriveGSM_ZSW1;
	nStatusExpected 	: WORD;
END_VAR
TEST('Set State S3');

//Arrange
fbFSM.eState := E_ProfidriveGSM_State.S3_SwitchedOn;

stStatusExpected.b0_ReadyToSwitchOn 		:= TRUE;				
stStatusExpected.b1_ReadyForOperation 		:= TRUE;				
stStatusExpected.b2_OperationEnabled 		:= FALSE;
stStatusExpected.b6_SwitchingOnInhibited 	:= FALSE;
MEMCPY(ADR(nStatusExpected), ADR(stStatusExpected), 2);

//Act
fbFSM();

//Assert
IF (nStatusExpected <> fbFSM.nStatus) THEN
	AssertEquals_BOOL(stStatusExpected.b0_ReadyToSwitchOn, fbFSM.stZSW1.b0_ReadyToSwitchOn, 'b0_ReadyToSwitchOn: AssertEquals not returning expected value');
	AssertEquals_BOOL(stStatusExpected.b1_ReadyForOperation, fbFSM.stZSW1.b1_ReadyForOperation, 'b1_ReadyForOperation: AssertEquals not returning expected value');
	AssertEquals_BOOL(stStatusExpected.b2_OperationEnabled, fbFSM.stZSW1.b2_OperationEnabled, 'b2_OperationEnabled: AssertEquals not returning expected value');	
	AssertEquals_BOOL(stStatusExpected.b6_SwitchingOnInhibited, fbFSM.stZSW1.b6_SwitchingOnInhibited, 'b6_SwitchingOnInhibited: AssertEquals not returning expected value');	
END_IF

TEST_FINISHED();
END_METHOD

METHOD TestState_S4 : BOOL
VAR
	fbFSM 				: FB_ProfidriveGSM;
	stStatusExpected	: ST_ProfiidriveGSM_ZSW1;
	nStatusExpected 	: WORD;
END_VAR
TEST('Set State S4');

//Arrange
fbFSM.eState := E_ProfidriveGSM_State.S4_Operation;

stStatusExpected.b0_ReadyToSwitchOn 		:= TRUE;				
stStatusExpected.b1_ReadyForOperation 		:= TRUE;				
stStatusExpected.b2_OperationEnabled 		:= TRUE;
stStatusExpected.b6_SwitchingOnInhibited 	:= FALSE;
MEMCPY(ADR(nStatusExpected), ADR(stStatusExpected), 2);

//Act
fbFSM();

//Assert
IF (nStatusExpected <> fbFSM.nStatus) THEN
	AssertEquals_BOOL(stStatusExpected.b0_ReadyToSwitchOn, fbFSM.stZSW1.b0_ReadyToSwitchOn, 'b0_ReadyToSwitchOn: AssertEquals not returning expected value');
	AssertEquals_BOOL(stStatusExpected.b1_ReadyForOperation, fbFSM.stZSW1.b1_ReadyForOperation, 'b1_ReadyForOperation: AssertEquals not returning expected value');
	AssertEquals_BOOL(stStatusExpected.b2_OperationEnabled, fbFSM.stZSW1.b2_OperationEnabled, 'b2_OperationEnabled: AssertEquals not returning expected value');	
	AssertEquals_BOOL(stStatusExpected.b6_SwitchingOnInhibited, fbFSM.stZSW1.b6_SwitchingOnInhibited, 'b6_SwitchingOnInhibited: AssertEquals not returning expected value');	
END_IF

TEST_FINISHED();
END_METHOD

METHOD TestState_S51 : BOOL
VAR
	fbFSM 				: FB_ProfidriveGSM;
	stStatusExpected	: ST_ProfiidriveGSM_ZSW1;
	nStatusExpected 	: WORD;
END_VAR
TEST('Set State S51');

//Arrange
fbFSM.eState := E_ProfidriveGSM_State.S51_RampStop;

stStatusExpected.b0_ReadyToSwitchOn 		:= TRUE;				
stStatusExpected.b1_ReadyForOperation 		:= TRUE;				
stStatusExpected.b2_OperationEnabled 		:= FALSE;
stStatusExpected.b6_SwitchingOnInhibited 	:= FALSE;
MEMCPY(ADR(nStatusExpected), ADR(stStatusExpected), 2);

//Act
fbFSM();

//Assert
IF (nStatusExpected <> fbFSM.nStatus) THEN
	AssertEquals_BOOL(stStatusExpected.b0_ReadyToSwitchOn, fbFSM.stZSW1.b0_ReadyToSwitchOn, 'b0_ReadyToSwitchOn: AssertEquals not returning expected value');
	AssertEquals_BOOL(stStatusExpected.b1_ReadyForOperation, fbFSM.stZSW1.b1_ReadyForOperation, 'b1_ReadyForOperation: AssertEquals not returning expected value');
	AssertEquals_BOOL(stStatusExpected.b2_OperationEnabled, fbFSM.stZSW1.b2_OperationEnabled, 'b2_OperationEnabled: AssertEquals not returning expected value');	
	AssertEquals_BOOL(stStatusExpected.b6_SwitchingOnInhibited, fbFSM.stZSW1.b6_SwitchingOnInhibited, 'b6_SwitchingOnInhibited: AssertEquals not returning expected value');	
END_IF

TEST_FINISHED();
END_METHOD

METHOD TestState_S52 : BOOL
VAR
	fbFSM 				: FB_ProfidriveGSM;
	stStatusExpected	: ST_ProfiidriveGSM_ZSW1;
	nStatusExpected 	: WORD;
END_VAR
TEST('Set State S52');

//Arrange
fbFSM.eState := E_ProfidriveGSM_State.S52_QuickStop;

stStatusExpected.b0_ReadyToSwitchOn 		:= TRUE;				
stStatusExpected.b1_ReadyForOperation 		:= TRUE;				
stStatusExpected.b2_OperationEnabled 		:= FALSE;
stStatusExpected.b6_SwitchingOnInhibited 	:= FALSE;
MEMCPY(ADR(nStatusExpected), ADR(stStatusExpected), 2);

//Act
fbFSM();

//Assert
IF (nStatusExpected <> fbFSM.nStatus) THEN
	AssertEquals_BOOL(stStatusExpected.b0_ReadyToSwitchOn, fbFSM.stZSW1.b0_ReadyToSwitchOn, 'b0_ReadyToSwitchOn: AssertEquals not returning expected value');
	AssertEquals_BOOL(stStatusExpected.b1_ReadyForOperation, fbFSM.stZSW1.b1_ReadyForOperation, 'b1_ReadyForOperation: AssertEquals not returning expected value');
	AssertEquals_BOOL(stStatusExpected.b2_OperationEnabled, fbFSM.stZSW1.b2_OperationEnabled, 'b2_OperationEnabled: AssertEquals not returning expected value');	
	AssertEquals_BOOL(stStatusExpected.b6_SwitchingOnInhibited, fbFSM.stZSW1.b6_SwitchingOnInhibited, 'b6_SwitchingOnInhibited: AssertEquals not returning expected value');	
END_IF

TEST_FINISHED();
END_METHOD

METHOD TestTransitions_S0 : BOOL
VAR
	fbFSM 				: FB_ProfidriveGSM;
	stStatusExpected	: ST_ProfiidriveGSM_ZSW1;
	nStatusExpected 	: WORD;
END_VAR
TEST('Transition S0>S0');

//Arrange
fbFSM.bPowerOn := FALSE;
fbFSM.eState := E_ProfidriveGSM_State.S0_Disabled;

//Act
fbFSM();

//Assert
AssertEquals_INT(E_ProfidriveGSM_State.S0_Disabled, fbFSM.eState, 'eState: AssertEquals not returning expected value');

TEST_FINISHED();


TEST('Transition S0>S1');

//Arrange
fbFSM.bPowerOn := TRUE;
fbFSM.eState := E_ProfidriveGSM_State.S0_Disabled;

//Act
fbFSM();

//Assert
AssertEquals_INT(E_ProfidriveGSM_State.S1_SwitchingOnInhibited, fbFSM.eState, 'eState: AssertEquals not returning expected value');

TEST_FINISHED();
END_METHOD

METHOD TestTransitions_S1 : BOOL
VAR
	fbFSM 				: FB_ProfidriveGSM;
	stStatusExpected	: ST_ProfiidriveGSM_ZSW1;
	nStatusExpected 	: WORD;
END_VAR
TEST('Transition S1>S2');

//Arrange
fbFSM.bPowerOn := TRUE;
fbFSM.eState := E_ProfidriveGSM_State.S1_SwitchingOnInhibited;

fbFSM.stSTW1.b0_On 				:= FALSE;
fbFSM.stSTW1.b1_CoastStop 		:= TRUE;
fbFSM.stSTW1.b2_QuickStop 		:= TRUE;

//Act
fbFSM();

//Assert
AssertEquals_INT(E_ProfidriveGSM_State.S2_ReadyForSwitchingOn, fbFSM.eState, 'eState: AssertEquals not returning expected value');

TEST_FINISHED();
END_METHOD

METHOD TestTransitions_S2 : BOOL
VAR
	fbFSM 				: FB_ProfidriveGSM;
	stStatusExpected	: ST_ProfiidriveGSM_ZSW1;
	nStatusExpected 	: WORD;
END_VAR
TEST('Transition S2>S1 Case_1');

//Arrange
fbFSM.bPowerOn := TRUE;
fbFSM.eState := E_ProfidriveGSM_State.S2_ReadyForSwitchingOn;

fbFSM.stSTW1.b0_On 				:= TRUE;
fbFSM.stSTW1.b1_CoastStop 		:= FALSE;
fbFSM.stSTW1.b2_QuickStop 		:= TRUE;

//Act
fbFSM();

//Assert
AssertEquals_INT(E_ProfidriveGSM_State.S1_SwitchingOnInhibited, fbFSM.eState, 'eState: AssertEquals not returning expected value');

TEST_FINISHED();


TEST('Transition S2>S1 Case_2');

//Arrange
fbFSM.bPowerOn := TRUE;
fbFSM.eState := E_ProfidriveGSM_State.S2_ReadyForSwitchingOn;

fbFSM.stSTW1.b0_On 				:= TRUE;
fbFSM.stSTW1.b1_CoastStop 		:= TRUE;
fbFSM.stSTW1.b2_QuickStop 		:= FALSE;

//Act
fbFSM();

//Assert
AssertEquals_INT(E_ProfidriveGSM_State.S1_SwitchingOnInhibited, fbFSM.eState, 'eState: AssertEquals not returning expected value');

TEST_FINISHED();


TEST('Transition S2 Still');

//Arrange
fbFSM.bPowerOn := TRUE;
fbFSM.eState := E_ProfidriveGSM_State.S2_ReadyForSwitchingOn;

fbFSM.stSTW1.b0_On 				:= FALSE;
fbFSM.stSTW1.b1_CoastStop 		:= TRUE;
fbFSM.stSTW1.b2_QuickStop 		:= TRUE;

//Act
fbFSM();

//Assert
AssertEquals_INT(E_ProfidriveGSM_State.S2_ReadyForSwitchingOn, fbFSM.eState, 'eState: AssertEquals not returning expected value');

TEST_FINISHED();


TEST('Transition S2>S3');

//Arrange
fbFSM.bPowerOn := TRUE;
fbFSM.eState := E_ProfidriveGSM_State.S2_ReadyForSwitchingOn;

fbFSM.stSTW1.b0_On 				:= TRUE;
fbFSM.stSTW1.b1_CoastStop 		:= TRUE;
fbFSM.stSTW1.b2_QuickStop 		:= TRUE;

//Act
fbFSM();

//Assert
AssertEquals_INT(E_ProfidriveGSM_State.S3_SwitchedOn, fbFSM.eState, 'eState: AssertEquals not returning expected value');

TEST_FINISHED();
END_METHOD

METHOD TestTransitions_S3 : BOOL
VAR
	fbFSM 				: FB_ProfidriveGSM;
	stStatusExpected	: ST_ProfiidriveGSM_ZSW1;
	nStatusExpected 	: WORD;
END_VAR
TEST('Transition S3>S1 Case_1');

//Arrange
fbFSM.bPowerOn := TRUE;
fbFSM.eState := E_ProfidriveGSM_State.S3_SwitchedOn;

fbFSM.stSTW1.b0_On 				:= TRUE;
fbFSM.stSTW1.b1_CoastStop 		:= FALSE;
fbFSM.stSTW1.b2_QuickStop 		:= TRUE;

//Act
fbFSM();

//Assert
AssertEquals_INT(E_ProfidriveGSM_State.S1_SwitchingOnInhibited, fbFSM.eState, 'eState: AssertEquals not returning expected value');

TEST_FINISHED();


TEST('Transition S3>S1 Case_2');

//Arrange
fbFSM.bPowerOn := TRUE;
fbFSM.eState := E_ProfidriveGSM_State.S3_SwitchedOn;

fbFSM.stSTW1.b0_On 				:= TRUE;
fbFSM.stSTW1.b1_CoastStop 		:= TRUE;
fbFSM.stSTW1.b2_QuickStop 		:= FALSE;

//Act
fbFSM();

//Assert
AssertEquals_INT(E_ProfidriveGSM_State.S1_SwitchingOnInhibited, fbFSM.eState, 'eState: AssertEquals not returning expected value');

TEST_FINISHED();


TEST('Transition S3 Still');

//Arrange
fbFSM.bPowerOn := TRUE;
fbFSM.eState := E_ProfidriveGSM_State.S3_SwitchedOn;

fbFSM.stSTW1.b0_On 				:= TRUE;
fbFSM.stSTW1.b1_CoastStop 		:= TRUE;
fbFSM.stSTW1.b2_QuickStop 		:= TRUE;
fbFSM.stSTW1.b3_EnableOperation  := FALSE;

//Act
fbFSM();

//Assert
AssertEquals_INT(E_ProfidriveGSM_State.S3_SwitchedOn, fbFSM.eState, 'eState: AssertEquals not returning expected value');

TEST_FINISHED();


TEST('Transition S3>S2');

//Arrange
fbFSM.bPowerOn := TRUE;
fbFSM.eState := E_ProfidriveGSM_State.S3_SwitchedOn;

fbFSM.stSTW1.b0_On 				:= FALSE;
fbFSM.stSTW1.b1_CoastStop 		:= TRUE;
fbFSM.stSTW1.b2_QuickStop 		:= TRUE;

//Act
fbFSM();

//Assert
AssertEquals_INT(E_ProfidriveGSM_State.S2_ReadyForSwitchingOn, fbFSM.eState, 'eState: AssertEquals not returning expected value');

TEST_FINISHED();


TEST('Transition S3>S4');

//Arrange
fbFSM.bPowerOn := TRUE;
fbFSM.eState := E_ProfidriveGSM_State.S3_SwitchedOn;

fbFSM.stSTW1.b0_On 				:= TRUE;
fbFSM.stSTW1.b1_CoastStop 		:= TRUE;
fbFSM.stSTW1.b2_QuickStop 		:= TRUE;
fbFSM.stSTW1.b3_EnableOperation  := TRUE;

//Act
fbFSM();

//Assert
AssertEquals_INT(E_ProfidriveGSM_State.S4_Operation, fbFSM.eState, 'eState: AssertEquals not returning expected value');

TEST_FINISHED();
END_METHOD

METHOD TestTransitions_S4 : BOOL
VAR
	fbFSM 				: FB_ProfidriveGSM;
	stStatusExpected	: ST_ProfiidriveGSM_ZSW1;
	nStatusExpected 	: WORD;
END_VAR
TEST('Transition S4>S1');

//Arrange
fbFSM.bPowerOn := TRUE;
fbFSM.eState := E_ProfidriveGSM_State.S4_Operation;

fbFSM.stSTW1.b0_On 				:= FALSE;
fbFSM.stSTW1.b1_CoastStop 		:= FALSE;
fbFSM.stSTW1.b2_QuickStop 		:= FALSE;

//Act
fbFSM();

//Assert
AssertEquals_INT(E_ProfidriveGSM_State.S1_SwitchingOnInhibited, fbFSM.eState, 'eState: AssertEquals not returning expected value');

TEST_FINISHED();


TEST('Transition S4>S52');

//Arrange
fbFSM.bPowerOn := TRUE;
fbFSM.eState := E_ProfidriveGSM_State.S4_Operation;

fbFSM.stSTW1.b0_On 				:= FALSE;
fbFSM.stSTW1.b1_CoastStop 		:= TRUE;
fbFSM.stSTW1.b2_QuickStop 		:= FALSE;

//Act
fbFSM();

//Assert
AssertEquals_INT(E_ProfidriveGSM_State.S52_QuickStop, fbFSM.eState, 'eState: AssertEquals not returning expected value');

TEST_FINISHED();


TEST('Transition S4>S51');

//Arrange
fbFSM.bPowerOn := TRUE;
fbFSM.eState := E_ProfidriveGSM_State.S4_Operation;

fbFSM.stSTW1.b0_On 				:= FALSE;
fbFSM.stSTW1.b1_CoastStop 		:= TRUE;
fbFSM.stSTW1.b2_QuickStop 		:= TRUE;
fbFSM.stSTW1.b3_EnableOperation 	:= FALSE;

//Act
fbFSM();

//Assert
AssertEquals_INT(E_ProfidriveGSM_State.S51_RampStop, fbFSM.eState, 'eState: AssertEquals not returning expected value');

TEST_FINISHED();


TEST('Transition S4>S3');

//Arrange
fbFSM.bPowerOn := TRUE;
fbFSM.eState := E_ProfidriveGSM_State.S4_Operation;

fbFSM.stSTW1.b0_On 				:= TRUE;
fbFSM.stSTW1.b1_CoastStop 		:= TRUE;
fbFSM.stSTW1.b2_QuickStop 		:= TRUE;
fbFSM.stSTW1.b3_EnableOperation 	:= FALSE;

//Act
fbFSM();

//Assert
AssertEquals_INT(E_ProfidriveGSM_State.S3_SwitchedOn, fbFSM.eState, 'eState: AssertEquals not returning expected value');

TEST_FINISHED();
END_METHOD

METHOD TestTransitions_S51 : BOOL
VAR
	fbFSM 				: FB_ProfidriveGSM;
	stStatusExpected	: ST_ProfiidriveGSM_ZSW1;
	nStatusExpected 	: WORD;
END_VAR
TEST('Transition S51 Still');

//Arrange
fbFSM.bPowerOn := TRUE;
fbFSM.eState := E_ProfidriveGSM_State.S51_RampStop;

fbFSM.bStandstill					:= FALSE;
fbFSM.stSTW1.b0_On 				:= FALSE;
fbFSM.stSTW1.b1_CoastStop 		:= TRUE;
fbFSM.stSTW1.b2_QuickStop 		:= TRUE;
fbFSM.stSTW1.b3_EnableOperation 	:= TRUE;

//Act
fbFSM();

//Assert
AssertEquals_INT(E_ProfidriveGSM_State.S51_RampStop, fbFSM.eState, 'eState: AssertEquals not returning expected value');

TEST_FINISHED();


TEST('Transition S51>S1');

//Arrange
fbFSM.bPowerOn := TRUE;
fbFSM.eState := E_ProfidriveGSM_State.S51_RampStop;

fbFSM.bStandstill					:= FALSE;
fbFSM.stSTW1.b0_On 				:= FALSE;
fbFSM.stSTW1.b1_CoastStop 		:= FALSE;
fbFSM.stSTW1.b2_QuickStop 		:= FALSE;
fbFSM.stSTW1.b3_EnableOperation 	:= FALSE;

//Act
fbFSM();

